C05459=1092.493,135.328,434.820,176.042,18.380,152.701
C05460=1092.487,135.079,434.840,176.041,18.379,152.701
C05461=1092.482,134.830,434.859,176.038,18.378,152.701
C05462=1092.476,134.580,434.880,176.035,18.377,152.702
C05463=1092.470,134.332,434.900,176.032,18.376,152.702
C05464=1092.465,134.082,434.919,176.030,18.376,152.702
C05465=1092.459,133.833,434.940,176.027,18.375,152.703
C05466=1092.454,133.585,434.959,176.025,18.374,152.703
C05467=1092.449,133.335,434.979,176.022,18.372,152.703
C05468=1092.443,133.086,434.999,176.020,18.372,152.703
C05469=1092.437,132.837,435.018,176.017,18.371,152.704
C05470=1092.432,132.588,435.039,176.015,18.370,152.704
C05471=1092.426,132.338,435.058,176.012,18.368,152.704
C05472=1092.420,132.090,435.078,176.010,18.368,152.704
C05473=1092.415,131.841,435.099,176.007,18.367,152.705
C05474=1092.409,131.591,435.118,176.004,18.366,152.705
C05475=1092.403,131.342,435.138,176.001,18.365,152.705
C05476=1092.398,131.093,435.157,175.999,18.364,152.706
C05477=1092.392,130.844,435.177,175.997,18.363,152.706
C05478=1092.386,130.595,435.196,175.994,18.362,152.706
C05479=1092.381,130.345,435.217,175.992,18.361,152.706
C05480=1092.375,130.096,435.236,175.989,18.360,152.707
C05481=1092.369,129.847,435.256,175.987,18.359,152.707
C05482=1092.363,129.598,435.275,175.984,18.358,152.707
C05483=1092.358,129.349,435.295,175.982,18.357,152.707
C05484=1092.352,129.100,435.314,175.979,18.356,152.708
C05485=1092.347,128.850,435.335,175.976,18.355,152.708
C05486=1092.341,128.601,435.354,175.975,18.355,152.708
C05487=1092.335,128.352,435.374,175.972,18.353,152.708
C05488=1092.328,128.076,435.395,175.969,18.352,152.709
C05489=1092.322,127.799,435.418,175.966,18.352,152.709
C05490=1092.316,127.522,435.439,175.963,18.351,152.709
C05491=1092.310,127.246,435.460,175.961,18.349,152.710
C05492=1092.304,126.997,435.480,175.958,18.348,152.710
C05493=1092.298,126.748,435.499,175.955,18.347,152.710
C05494=1092.292,126.499,435.519,175.953,18.347,152.710
C05495=1092.287,126.249,435.539,175.950,18.345,152.711
C05496=1092.282,126.000,435.558,175.948,18.344,152.711
C05497=1092.276,125.751,435.578,175.946,18.344,152.711
C05498=1092.270,125.502,435.597,175.943,18.343,152.711
C05499=1092.265,125.253,435.617,175.940,18.341,152.712
C05500=1092.259,125.003,435.636,175.938,18.340,152.712
C05501=1092.253,124.754,435.656,175.936,18.339,152.712
C05502=1092.247,124.505,435.675,175.933,18.338,152.712
C05503=1092.242,124.255,435.694,175.930,18.337,152.713
C05504=1092.236,124.007,435.714,175.928,18.336,152.713
C05505=1092.231,123.758,435.733,175.926,18.335,152.713
C05506=1092.225,123.508,435.752,175.923,18.334,152.713
C05507=1092.219,123.259,435.772,175.920,18.333,152.714
C05508=1092.214,123.010,435.791,175.918,18.332,152.714
C05509=1092.208,122.760,435.811,175.916,18.331,152.714
C05510=1092.203,122.512,435.830,175.913,18.330,152.714
C05511=1092.198,122.262,435.849,175.911,18.329,152.715
C05512=1092.192,122.013,435.869,175.908,18.328,152.715
C05513=1092.186,121.763,435.888,175.906,18.327,152.715
C05514=1092.180,121.515,435.908,175.904,18.326,152.715
C05515=1092.175,121.266,435.927,175.901,18.324,152.715
C05516=1092.169,121.016,435.946,175.899,18.323,152.716
C05517=1092.164,120.767,435.965,175.897,18.323,152.716
C05518=1092.158,120.518,435.985,175.894,18.322,152.716
C05519=1092.152,120.268,436.004,175.891,18.320,152.716
C05520=1092.147,120.019,436.023,175.890,18.319,152.717
C05521=1092.142,119.770,436.042,175.887,18.318,152.717
C05522=1092.136,119.521,436.062,175.884,18.317,152.717
C05523=1092.130,119.272,436.081,175.881,18.316,152.717
C05524=1092.125,119.023,436.100,175.880,18.315,152.717
C05525=1092.119,118.774,436.119,175.877,18.314,152.718
C05526=1092.113,118.524,436.138,175.874,18.313,152.718
C05527=1092.108,118.275,436.157,175.872,18.312,152.718
C05528=1092.103,118.026,436.177,175.870,18.310,152.718
C05529=1092.097,117.777,436.196,175.867,18.309,152.719
C05530=1092.091,117.527,436.214,175.865,18.309,152.719
C05531=1092.085,117.279,436.233,175.863,18.307,152.719
C05532=1092.080,117.029,436.253,175.860,18.306,152.719
C05533=1092.074,116.780,436.272,175.858,18.305,152.719
C05534=1092.069,116.531,436.291,175.855,18.304,152.720
C05535=1092.063,116.282,436.310,175.853,18.303,152.720
C05536=1092.058,116.032,436.329,175.851,18.302,152.720
C05537=1092.053,115.784,436.348,175.848,18.300,152.720
C05538=1092.047,115.534,436.367,175.846,18.299,152.721
C05539=1092.041,115.284,436.386,175.844,18.299,152.721
C05540=1092.036,115.035,436.405,175.841,18.297,152.721
C05541=1092.031,114.786,436.424,175.838,18.296,152.721
C05542=1092.025,114.536,436.443,175.837,18.295,152.721
C05543=1092.019,114.288,436.461,175.834,18.294,152.722
C05544=1092.013,114.039,436.481,175.831,18.293,152.722
C05545=1092.008,113.789,436.500,175.829,18.292,152.722
C05546=1092.003,113.540,436.519,175.827,18.290,152.722
C05547=1091.997,113.291,436.537,175.824,18.289,152.722
C05548=1091.991,113.041,436.556,175.822,18.289,152.723
C05549=1091.986,112.793,436.575,175.820,18.287,152.723
C05550=1091.980,112.543,436.594,175.817,18.286,152.723
C05551=1091.974,112.294,436.613,175.815,18.285,152.723
C05552=1091.968,112.017,436.634,175.813,18.284,152.723
C05553=1091.962,111.741,436.654,175.810,18.283,152.724
C05554=1091.956,111.465,436.676,175.807,18.281,152.724
C05555=1091.949,111.187,436.696,175.805,18.280,152.724
C05556=1091.943,110.939,436.715,175.802,18.279,152.724
C05557=1091.938,110.690,436.734,175.800,18.278,152.725
C05558=1091.932,110.439,436.752,175.798,18.276,152.725
C05559=1091.926,110.191,436.771,175.795,18.275,152.725
C05560=1091.921,109.942,436.790,175.793,18.274,152.725
C05561=1091.915,109.692,436.809,175.790,18.273,152.725
C05562=1091.910,109.443,436.827,175.788,18.272,152.726
C05563=1091.904,109.194,436.846,175.786,18.271,152.726
C05564=1091.898,108.945,436.864,175.783,18.270,152.726
C05565=1091.893,108.695,436.883,175.781,18.268,152.726
C05566=1091.887,108.446,436.902,175.779,18.268,152.726
C05567=1091.881,108.197,436.920,175.776,18.266,152.727
C05568=1091.876,107.947,436.939,175.774,18.265,152.727
C05569=1091.869,107.698,436.958,175.772,18.264,152.727
C05570=1091.865,107.449,436.976,175.769,18.263,152.727
C05571=1091.858,107.200,436.994,175.767,18.262,152.727
C05572=1091.853,106.951,437.013,175.765,18.260,152.727
C05573=1091.848,106.701,437.032,175.762,18.259,152.728
C05574=1091.842,106.453,437.050,175.760,18.258,152.728
C05575=1091.836,106.203,437.069,175.758,18.257,152.728
C05576=1091.830,105.953,437.087,175.755,18.255,152.728
C05577=1091.825,105.705,437.106,175.753,18.255,152.728
C05578=1091.819,105.455,437.124,175.751,18.253,152.729
C05579=1091.814,105.206,437.143,175.749,18.253,152.729
C05580=1091.808,104.956,437.161,175.746,18.251,152.729
C05581=1091.803,104.708,437.180,175.744,18.250,152.729
C05582=1091.797,104.458,437.198,175.742,18.249,152.729
C05583=1091.791,104.209,437.217,175.739,18.248,152.730
C05584=1091.786,103.959,437.235,175.737,18.246,152.730
C05585=1091.780,103.711,437.253,175.735,18.245,152.730
C05586=1091.775,103.461,437.272,175.732,18.244,152.730
C05587=1091.769,103.212,437.290,175.730,18.243,152.730
C05588=1091.764,102.962,437.309,175.728,18.242,152.730
C05589=1091.758,102.714,437.327,175.726,18.240,152.731
C05590=1091.752,102.464,437.345,175.724,18.239,152.731
C05591=1091.746,102.215,437.364,175.721,18.238,152.731
C05592=1091.741,101.965,437.382,175.718,18.237,152.731
C05593=1091.736,101.716,437.400,175.717,18.236,152.731
C05594=1091.730,101.467,437.419,175.714,18.234,152.731
C05595=1091.724,101.218,437.437,175.712,18.233,152.732
C05596=1091.718,100.969,437.455,175.710,18.232,152.732
C05597=1091.713,100.719,437.473,175.707,18.231,152.732
C05598=1091.707,100.470,437.491,175.705,18.229,152.732
C05599=1091.701,100.221,437.510,175.703,18.228,152.732
C05600=1091.696,99.971,437.528,175.701,18.227,152.733
C05601=1091.690,99.722,437.546,175.699,18.226,152.733
C05602=1091.684,99.473,437.564,175.696,18.225,152.733
C05603=1091.679,99.224,437.583,175.694,18.223,152.733
C05604=1091.673,98.974,437.601,175.691,18.222,152.733
C05605=1091.667,98.725,437.619,175.690,18.221,152.733
C05606=1091.662,98.475,437.637,175.687,18.220,152.733
C05607=1091.656,98.226,437.655,175.685,18.219,152.734
C05608=1091.650,97.977,437.674,175.683,18.217,152.734
C05609=1091.644,97.728,437.691,175.680,18.216,152.734
C05610=1091.639,97.478,437.710,175.678,18.215,152.734
C05611=1091.633,97.230,437.728,175.676,18.214,152.734
C05612=1091.627,96.980,437.746,175.673,18.212,152.735
C05613=1091.622,96.731,437.764,175.672,18.211,152.735
C05614=1091.617,96.482,437.782,175.669,18.210,152.735
C05615=1091.611,96.232,437.800,175.667,18.209,152.735
C05616=1091.604,95.955,437.820,175.665,18.208,152.735
C05617=1091.598,95.679,437.840,175.662,18.206,152.735
C05618=1091.592,95.403,437.860,175.659,18.205,152.736
C05619=1091.586,95.126,437.879,175.657,18.203,152.736
C05620=1091.580,94.876,437.898,175.655,18.202,152.736
C05621=1091.574,94.628,437.916,175.653,18.200,152.736
C05622=1091.568,94.378,437.934,175.650,18.199,152.736
C05623=1091.563,94.129,437.952,175.648,18.198,152.736
C05624=1091.558,93.880,437.970,175.646,18.197,152.736
C05625=1091.552,93.630,437.988,175.644,18.196,152.737
C05626=1091.546,93.381,438.005,175.642,18.194,152.737
C05627=1091.541,93.132,438.023,175.639,18.193,152.737
C05628=1091.535,92.882,438.041,175.637,18.192,152.737
C05629=1091.530,92.633,438.060,175.635,18.190,152.737
C05630=1091.524,92.384,438.077,175.633,18.190,152.737
C05631=1091.518,92.135,438.095,175.631,18.188,152.738
C05632=1091.512,91.886,438.113,175.628,18.186,152.738
C05633=1091.507,91.637,438.130,175.626,18.185,152.738
C05634=1091.502,91.386,438.149,175.624,18.184,152.738
C05635=1091.496,91.137,438.166,175.622,18.183,152.738
C05636=1091.491,90.888,438.184,175.620,18.181,152.738
C05637=1091.484,90.639,438.202,175.618,18.180,152.738
C05638=1091.479,90.390,438.219,175.615,18.179,152.738
C05639=1091.473,90.140,438.237,175.613,18.178,152.739
C05640=1091.467,89.891,438.255,175.611,18.177,152.739
C05641=1091.462,89.642,438.272,175.609,18.175,152.739
C05642=1091.456,89.392,438.290,175.607,18.174,152.739
C05643=1091.450,89.143,438.308,175.604,18.173,152.739
C05644=1091.445,88.894,438.325,175.602,18.172,152.739
C05645=1091.438,88.644,438.343,175.600,18.170,152.740
C05646=1091.433,88.395,438.361,175.598,18.168,152.740
C05647=1091.427,88.146,438.379,175.596,18.167,152.740
C05648=1091.421,87.896,438.396,175.593,18.166,152.740
C05649=1091.416,87.647,438.414,175.591,18.165,152.740
C05650=1091.411,87.398,438.431,175.589,18.163,152.740
C05651=1091.404,87.148,438.449,175.587,18.162,152.740
C05652=1091.399,86.899,438.466,175.585,18.161,152.740
C05653=1091.393,86.650,438.484,175.582,18.159,152.741
C05654=1091.387,86.400,438.502,175.580,18.159,152.741
C05655=1091.382,86.151,438.519,175.578,18.157,152.741
C05656=1091.376,85.902,438.537,175.576,18.156,152.741
C05657=1091.371,85.653,438.555,175.574,18.154,152.741
C05658=1091.365,85.403,438.572,175.572,18.153,152.741
C05659=1091.359,85.154,438.589,175.570,18.152,152.741
C05660=1091.354,84.905,438.607,175.568,18.150,152.742
C05661=1091.348,84.656,438.625,175.566,18.149,152.742
C05662=1091.342,84.406,438.642,175.563,18.148,152.742
C05663=1091.337,84.156,438.659,175.561,18.147,152.742
C05664=1091.332,83.907,438.677,175.559,18.145,152.742
C05665=1091.325,83.658,438.694,175.557,18.144,152.742
C05666=1091.319,83.409,438.712,175.555,18.142,152.742
C05667=1091.314,83.159,438.729,175.553,18.141,152.742
C05668=1091.308,82.910,438.746,175.550,18.140,152.743
C05669=1091.303,82.661,438.764,175.549,18.139,152.743
C05670=1091.297,82.411,438.782,175.546,18.137,152.743
C05671=1091.292,82.161,438.799,175.544,18.135,152.743
C05672=1091.286,81.912,438.816,175.542,18.134,152.743
C05673=1091.281,81.663,438.834,175.540,18.133,152.743
C05674=1091.275,81.414,438.851,175.538,18.132,152.743
C05675=1091.270,81.165,438.868,175.536,18.130,152.743
C05676=1091.263,80.915,438.885,175.534,18.129,152.743
C05677=1091.258,80.666,438.902,175.531,18.127,152.744
C05678=1091.252,80.417,438.920,175.530,18.126,152.744
C05679=1091.247,80.168,438.937,175.527,18.125,152.744
C05680=1091.240,79.891,438.957,175.525,18.123,152.744
C05681=1091.234,79.615,438.975,175.522,18.121,152.744
C05682=1091.228,79.338,438.995,175.521,18.120,152.744
C05683=1091.222,79.062,439.013,175.518,18.119,152.744
C05684=1091.216,78.812,439.031,175.516,18.117,152.744
C05685=1091.210,78.563,439.049,175.514,18.116,152.745
C05686=1091.205,78.313,439.066,175.512,18.114,152.745
C05687=1091.199,78.064,439.083,175.510,18.113,152.745
C05688=1091.193,77.815,439.100,175.507,18.112,152.745
C05689=1091.188,77.566,439.117,175.506,18.110,152.745
C05690=1091.183,77.316,439.134,175.503,18.109,152.745
C05691=1091.176,77.067,439.151,175.502,18.108,152.745
C05692=1091.171,76.817,439.168,175.499,18.106,152.745
C05693=1091.165,76.568,439.186,175.497,18.105,152.745
C05694=1091.159,76.319,439.202,175.495,18.103,152.746
C05695=1091.154,76.069,439.220,175.493,18.102,152.746
C05696=1091.148,75.820,439.236,175.491,18.101,152.746
C05697=1091.142,75.570,439.254,175.488,18.099,152.746
C05698=1091.136,75.321,439.271,175.487,18.098,152.746
C05699=1091.131,75.072,439.288,175.484,18.096,152.746
C05700=1091.125,74.822,439.304,175.483,18.095,152.746
C05701=1091.119,74.573,439.322,175.480,18.094,152.746
C05702=1091.114,74.324,439.339,175.478,18.093,152.746
C05703=1091.108,74.075,439.356,175.476,18.091,152.746
C05704=1091.103,73.825,439.373,175.475,18.089,152.747
C05705=1091.097,73.576,439.390,175.472,18.088,152.747
C05706=1091.091,73.326,439.407,175.470,18.087,152.747
C05707=1091.085,73.076,439.424,175.468,18.085,152.747
C05708=1091.080,72.827,439.441,175.466,18.084,152.747
C05709=1091.074,72.578,439.458,175.464,18.082,152.747
C05710=1091.068,72.329,439.475,175.462,18.081,152.747
C05711=1091.062,72.080,439.491,175.460,18.080,152.747
C05712=1091.057,71.830,439.508,175.458,18.078,152.747
C05713=1091.052,71.581,439.526,175.456,18.077,152.747
C05714=1091.046,71.332,439.542,175.454,18.075,152.748
C05715=1091.041,71.082,439.559,175.452,18.074,152.748
C05716=1091.034,70.833,439.576,175.450,18.073,152.748
C05717=1091.029,70.584,439.593,175.448,18.071,152.748
C05718=1091.024,70.334,439.610,175.446,18.070,152.748
C05719=1091.018,70.085,439.626,175.444,18.068,152.748
C05720=1091.012,69.836,439.643,175.442,18.067,152.748
C05721=1091.006,69.586,439.660,175.440,18.065,152.748
C05722=1091.001,69.336,439.677,175.438,18.064,152.748
C05723=1090.994,69.087,439.694,175.435,18.063,152.748
C05724=1090.989,68.837,439.711,175.434,18.061,152.749
C05725=1090.983,68.588,439.727,175.431,18.060,152.749
C05726=1090.978,68.338,439.744,175.430,18.058,152.749
C05727=1090.972,68.090,439.761,175.427,18.057,152.749
C05728=1090.967,67.840,439.778,175.426,18.056,152.749
C05729=1090.961,67.591,439.794,175.423,18.054,152.749
C05730=1090.955,67.341,439.810,175.422,18.053,152.749
C05731=1090.949,67.092,439.827,175.419,18.051,152.749
C05732=1090.943,66.843,439.844,175.418,18.050,152.749
C05733=1090.938,66.593,439.861,175.415,18.048,152.749
C05734=1090.932,66.344,439.877,175.414,18.047,152.749
C05735=1090.927,66.094,439.894,175.411,18.045,152.749
C05736=1090.921,65.845,439.910,175.410,18.044,152.750
C05737=1090.915,65.596,439.926,175.407,18.042,152.750
C05738=1090.909,65.347,439.944,175.406,18.041,152.750
C05739=1090.903,65.097,439.960,175.403,18.039,152.750
C05740=1090.898,64.848,439.977,175.402,18.038,152.750
C05741=1090.892,64.598,439.993,175.399,18.036,152.750
C05742=1090.886,64.349,440.010,175.398,18.035,152.750
C05743=1090.881,64.099,440.026,175.395,18.034,152.750
C05744=1090.874,63.823,440.045,175.394,18.033,152.750
C05745=1090.867,63.546,440.063,175.391,18.031,152.750
C05746=1090.862,63.270,440.081,175.389,18.029,152.750
C05747=1090.855,62.994,440.099,175.386,18.027,152.750
C05748=1090.850,62.744,440.116,175.385,18.026,152.751
C05749=1090.844,62.495,440.132,175.382,18.024,152.751
C05750=1090.838,62.245,440.148,175.381,18.023,152.751
C05751=1090.832,61.996,440.164,175.378,18.022,152.751
C05752=1090.826,61.747,440.181,175.377,18.020,152.751
C05753=1090.821,61.497,440.198,175.374,18.019,152.751
C05754=1090.815,61.248,440.214,175.373,18.017,152.751
C05755=1090.809,60.998,440.230,175.371,18.016,152.751
C05756=1090.803,60.749,440.246,175.369,18.014,152.751
C05757=1090.797,60.499,440.263,175.367,18.013,152.751
C05758=1090.792,60.250,440.279,175.365,18.012,152.751
C05759=1090.786,60.000,440.296,175.363,18.011,152.751
C05760=1090.780,59.751,440.312,175.360,18.009,152.752
C05761=1090.774,59.502,440.328,175.359,18.007,152.752
C05762=1090.768,59.252,440.344,175.357,18.006,152.752
C05763=1090.762,59.003,440.361,175.355,18.005,152.752
C05764=1090.757,58.753,440.378,175.353,18.003,152.752
C05765=1090.751,58.504,440.394,175.351,18.001,152.752
C05766=1090.745,58.255,440.410,175.349,18.000,152.752
C05767=1090.739,58.005,440.426,175.347,17.999,152.752
C05768=1090.733,57.756,440.443,175.345,17.997,152.752
C05769=1090.728,57.507,440.458,175.343,17.996,152.752
C05770=1090.723,57.257,440.475,175.341,17.994,152.752
C05771=1090.717,57.008,440.491,175.339,17.992,152.752
C05772=1090.711,56.758,440.507,175.338,17.991,152.752
C05773=1090.705,56.509,440.523,175.335,17.990,152.752
C05774=1090.699,56.260,440.540,175.334,17.988,152.752
C05775=1090.693,56.010,440.556,175.331,17.986,152.753
C05776=1090.688,55.760,440.571,175.330,17.985,152.753
C05777=1090.682,55.511,440.588,175.327,17.983,152.753
C05778=1090.677,55.262,440.604,175.326,17.982,152.753
C05779=1090.671,55.013,440.620,175.323,17.981,152.753
C05780=1090.665,54.763,440.637,175.322,17.979,152.753
C05781=1090.659,54.513,440.652,175.320,17.978,152.753
C05782=1090.653,54.264,440.669,175.318,17.976,152.753
C05783=1090.648,54.015,440.685,175.316,17.975,152.753
C05784=1090.642,53.766,440.701,175.314,17.973,152.753
C05785=1090.637,53.516,440.716,175.312,17.971,152.753
C05786=1090.631,53.267,440.732,175.310,17.970,152.753
C05787=1090.625,53.017,440.749,175.308,17.969,152.753
C05788=1090.620,52.767,440.765,175.306,17.967,152.753
C05789=1090.614,52.518,440.781,175.304,17.966,152.753
C05790=1090.608,52.269,440.797,175.303,17.964,152.753
C05791=1090.602,52.020,440.813,175.301,17.962,152.753
C05792=1090.597,51.770,440.829,175.299,17.961,152.754
C05793=1090.591,51.520,440.845,175.297,17.959,152.754
C05794=1090.585,51.271,440.861,175.295,17.958,152.754
C05795=1090.580,51.022,440.876,175.293,17.956,152.754
C05796=1090.574,50.773,440.893,175.291,17.955,152.754
C05797=1090.568,50.523,440.909,175.289,17.953,152.754
C05798=1090.562,50.273,440.925,175.287,17.952,152.754
C05799=1090.557,50.025,440.940,175.286,17.951,152.754
C05800=1090.551,49.775,440.956,175.283,17.949,152.754
C05801=1090.545,49.525,440.972,175.282,17.947,152.754
C05802=1090.539,49.276,440.988,175.280,17.945,152.754
C05803=1090.534,49.027,441.004,175.278,17.944,152.754
C05804=1090.528,48.777,441.020,175.276,17.942,152.754
C05805=1090.523,48.527,441.035,175.274,17.941,152.754
C05806=1090.517,48.278,441.052,175.272,17.939,152.754
C05807=1090.512,48.029,441.067,175.270,17.938,152.754
C05808=1090.506,47.752,441.085,175.268,17.936,152.754
C05809=1090.499,47.475,441.103,175.266,17.935,152.754
C05810=1090.493,47.198,441.120,175.264,17.933,152.754
C05811=1090.487,46.922,441.138,175.262,17.930,152.754
C05812=1090.481,46.672,441.153,175.260,17.929,152.754
C05813=1090.476,46.423,441.169,175.258,17.927,152.754
C05814=1090.470,46.173,441.185,175.256,17.926,152.754
C05815=1090.464,45.924,441.201,175.255,17.925,152.754
C05816=1090.459,45.675,441.216,175.253,17.923,152.755
C05817=1090.453,45.425,441.232,175.251,17.921,152.755
C05818=1090.447,45.175,441.248,175.249,17.920,152.755
C05819=1090.442,44.926,441.263,175.247,17.918,152.755
C05820=1090.436,44.677,441.279,175.245,17.917,152.755
C05821=1090.431,44.427,441.295,175.243,17.915,152.755
C05822=1090.425,44.178,441.311,175.242,17.913,152.755
C05823=1090.420,43.928,441.326,175.240,17.912,152.755
C05824=1090.414,43.679,441.343,175.238,17.910,152.755
C05825=1090.409,43.429,441.358,175.236,17.909,152.755
C05826=1090.402,43.180,441.373,175.234,17.907,152.755
C05827=1090.396,42.930,441.389,175.232,17.905,152.755
C05828=1090.391,42.681,441.404,175.230,17.904,152.755
C05829=1090.385,42.432,441.420,175.229,17.903,152.755
C05830=1090.380,42.182,441.436,175.227,17.901,152.755
C05831=1090.374,41.933,441.451,175.225,17.899,152.755
C05832=1090.368,41.684,441.467,175.223,17.897,152.755
C05833=1090.362,41.434,441.482,175.221,17.896,152.755
C05834=1090.357,41.184,441.498,175.220,17.895,152.755
C05835=1090.351,40.935,441.514,175.217,17.893,152.755
C05836=1090.345,40.685,441.529,175.216,17.892,152.755
C05837=1090.340,40.436,441.544,175.213,17.890,152.755
C05838=1090.334,40.187,441.560,175.212,17.888,152.755
C05839=1090.328,39.937,441.576,175.211,17.887,152.755
C05840=1090.322,39.688,441.590,175.208,17.885,152.755
C05841=1090.317,39.438,441.606,175.207,17.884,152.755
C05842=1090.312,39.189,441.622,175.204,17.882,152.755
C05843=1090.306,38.939,441.637,175.203,17.880,152.755
C05844=1090.299,38.690,441.652,175.201,17.879,152.755
C05845=1090.294,38.440,441.667,175.199,17.877,152.755
C05846=1090.288,38.191,441.684,175.198,17.876,152.755
C05847=1090.283,37.942,441.699,175.195,17.874,152.756
C05848=1090.277,37.692,441.714,175.194,17.872,152.756
C05849=1090.271,37.442,441.729,175.192,17.871,152.756
C05850=1090.266,37.193,441.744,175.190,17.869,152.756
C05851=1090.260,36.944,441.760,175.188,17.868,152.756
C05852=1090.254,36.694,441.776,175.186,17.866,152.756
C05853=1090.248,36.445,441.790,175.184,17.865,152.756
C05854=1090.243,36.195,441.806,175.183,17.863,152.756
C05855=1090.236,35.945,441.821,175.181,17.861,152.756
C05856=1090.231,35.697,441.837,175.179,17.860,152.756
C05857=1090.224,35.447,441.852,175.177,17.858,152.756
C05858=1090.219,35.198,441.867,175.175,17.857,152.756
C05859=1090.214,34.948,441.882,175.174,17.855,152.756
C05860=1090.207,34.698,441.897,175.171,17.854,152.756
C05861=1090.202,34.449,441.912,175.170,17.852,152.756
C05862=1090.196,34.199,441.927,175.169,17.851,152.756
C05863=1090.191,33.950,441.943,175.166,17.849,152.756
C05864=1090.184,33.701,441.958,175.165,17.847,152.756
C05865=1090.179,33.452,441.973,175.162,17.846,152.756
C05866=1090.174,33.202,441.989,175.161,17.844,152.756
C05867=1090.167,32.952,442.004,175.160,17.843,152.756
C05868=1090.162,32.703,442.019,175.157,17.841,152.756
C05869=1090.156,32.453,442.034,175.156,17.839,152.756
C05870=1090.151,32.204,442.049,175.154,17.838,152.756
C05871=1090.144,31.954,442.064,175.152,17.836,152.756
C05872=1090.138,31.677,442.081,175.150,17.834,152.756
C05873=1090.132,31.400,442.098,175.148,17.833,152.756
C05874=1090.126,31.124,442.114,175.146,17.831,152.756
C05875=1090.120,30.847,442.131,175.144,17.829,152.756
C05876=1090.113,30.598,442.146,175.142,17.827,152.756
C05877=1090.108,30.348,442.161,175.141,17.826,152.756
C05878=1090.102,30.099,442.176,175.138,17.824,152.756
C05879=1090.097,29.849,442.191,175.137,17.823,152.756
C05880=1090.090,29.600,442.206,175.135,17.821,152.756
C05881=1090.085,29.351,442.221,175.133,17.819,152.756
C05882=1090.079,29.101,442.236,175.131,17.818,152.756
C05883=1090.074,28.852,442.252,175.130,17.816,152.756
C05884=1090.068,28.602,442.266,175.128,17.814,152.756
C05885=1090.063,28.353,442.282,175.126,17.813,152.756
C05886=1090.056,28.103,442.297,175.125,17.812,152.756
C05887=1090.051,27.853,442.310,175.123,17.810,152.756
C05888=1090.045,27.604,442.326,175.121,17.808,152.757
C05889=1090.039,27.355,442.341,175.119,17.806,152.757
C05890=1090.033,27.105,442.356,175.117,17.805,152.756
C05891=1090.028,26.856,442.371,175.116,17.804,152.757
C05892=1090.021,26.606,442.386,175.114,17.802,152.757
C05893=1090.016,26.357,442.401,175.112,17.800,152.756
C05894=1090.010,26.107,442.416,175.110,17.799,152.757
C05895=1090.005,25.857,442.430,175.108,17.797,152.757
C05896=1089.999,25.607,442.445,175.107,17.796,152.757
C05897=1089.993,25.359,442.460,175.105,17.794,152.757
C05898=1089.987,25.109,442.475,175.103,17.792,152.757
C05899=1089.981,24.860,442.489,175.101,17.791,152.757
C05900=1089.975,24.610,442.505,175.100,17.789,152.757
C05901=1089.970,24.360,442.519,175.098,17.787,152.757
C05902=1089.963,24.111,442.534,175.096,17.786,152.757
C05903=1089.958,23.861,442.549,175.095,17.784,152.757
C05904=1089.953,23.613,442.563,175.093,17.782,152.757
C05905=1089.947,23.362,442.578,175.091,17.781,152.757
C05906=1089.941,23.113,442.593,175.090,17.780,152.757
C05907=1089.935,22.863,442.608,175.087,17.778,152.757
C05908=1089.929,22.614,442.622,175.086,17.776,152.757
C05909=1089.923,22.364,442.637,175.084,17.775,152.757
C05910=1089.918,22.115,442.652,175.082,17.773,152.757
C05911=1089.912,21.866,442.666,175.081,17.771,152.757
C05912=1089.906,21.616,442.681,175.078,17.770,152.757
C05913=1089.901,21.366,442.696,175.077,17.768,152.757
C05914=1089.895,21.117,442.711,175.075,17.766,152.757
C05915=1089.889,20.868,442.725,175.073,17.765,152.757
C05916=1089.884,20.618,442.739,175.072,17.763,152.757
C05917=1089.878,20.368,442.755,175.070,17.762,152.757
C05918=1089.872,20.119,442.769,175.068,17.759,152.757
C05919=1089.866,19.869,442.783,175.066,17.758,152.757
C05920=1089.860,19.620,442.798,175.065,17.757,152.757
C05921=1089.855,19.371,442.813,175.063,17.755,152.757
C05922=1089.849,19.121,442.827,175.061,17.754,152.757
C05923=1089.843,18.871,442.842,175.060,17.752,152.757
C05924=1089.837,18.622,442.857,175.058,17.750,152.757
C05925=1089.832,18.372,442.871,175.056,17.749,152.757
C05926=1089.826,18.123,442.885,175.055,17.747,152.757
C05927=1089.820,17.873,442.900,175.053,17.746,152.757
C05928=1089.814,17.624,442.914,175.051,17.744,152.757
C05929=1089.809,17.374,442.928,175.049,17.742,152.757
C05930=1089.803,17.125,442.944,175.048,17.741,152.757
C05931=1089.797,16.876,442.958,175.046,17.739,152.757
C05932=1089.791,16.625,442.972,175.044,17.738,152.757
C05933=1089.785,16.376,442.987,175.043,17.736,152.757
C05934=1089.780,16.127,443.001,175.040,17.734,152.757
C05935=1089.773,15.877,443.016,175.039,17.732,152.757
C05936=1089.768,15.602,443.031,175.037,17.731,152.757
C05937=1089.761,15.326,443.048,175.035,17.729,152.757
C05938=1089.755,15.051,443.063,175.033,17.727,152.757
C05939=1089.748,14.776,443.079,175.032,17.725,152.757
C05940=1089.743,14.527,443.094,175.029,17.723,152.757
C05941=1089.737,14.277,443.108,175.028,17.722,152.757
C05942=1089.731,14.028,443.123,175.026,17.721,152.757
C05943=1089.725,13.778,443.136,175.024,17.719,152.757
C05944=1089.719,13.528,443.151,175.023,17.717,152.757
C05945=1089.713,13.279,443.165,175.021,17.716,152.757
C05946=1089.708,13.029,443.179,175.020,17.714,152.757
C05947=1089.702,12.780,443.194,175.018,17.712,152.757
C05948=1089.696,12.530,443.208,175.016,17.711,152.757
C05949=1089.690,12.281,443.223,175.015,17.709,152.757
C05950=1089.684,12.031,443.237,175.012,17.707,152.757
C05951=1089.679,11.781,443.251,175.011,17.706,152.757
C05952=1089.672,11.533,443.265,175.009,17.705,152.757
C05953=1089.666,11.282,443.279,175.007,17.703,152.757
C05954=1089.660,11.033,443.293,175.006,17.701,152.757
C05955=1089.655,10.784,443.307,175.004,17.700,152.757
C05956=1089.649,10.533,443.322,175.003,17.698,152.757
C05957=1089.643,10.285,443.336,175.001,17.696,152.757
C05958=1089.638,10.035,443.350,174.999,17.695,152.757
C05959=1089.632,9.785,443.364,174.998,17.694,152.757
C05960=1089.626,9.536,443.379,174.995,17.691,152.757
C05961=1089.620,9.286,443.393,174.994,17.690,152.757
C05962=1089.615,9.037,443.407,174.992,17.689,152.757
C05963=1089.608,8.787,443.421,174.990,17.687,152.757
C05964=1089.602,8.538,443.435,174.989,17.685,152.757
C05965=1089.597,8.288,443.449,174.987,17.684,152.757
C05966=1089.591,8.039,443.463,174.986,17.682,152.757
C05967=1089.585,7.789,443.477,174.983,17.680,152.757
C05968=1089.579,7.539,443.491,174.982,17.679,152.757
C05969=1089.574,7.290,443.506,174.980,17.678,152.757
C05970=1089.567,7.041,443.519,174.978,17.675,152.757
C05971=1089.561,6.791,443.533,174.977,17.674,152.757
C05972=1089.556,6.541,443.547,174.975,17.672,152.757
C05973=1089.550,6.292,443.562,174.974,17.671,152.757
C05974=1089.545,6.043,443.576,174.972,17.669,152.757
C05975=1089.538,5.792,443.590,174.970,17.667,152.757
C05976=1089.533,5.543,443.604,174.969,17.666,152.757
C05977=1089.527,5.294,443.617,174.966,17.664,152.757
C05978=1089.521,5.045,443.632,174.965,17.663,152.757
C05979=1089.516,4.795,443.645,174.964,17.661,152.757
C05980=1089.509,4.545,443.660,174.962,17.659,152.757
C05981=1089.504,4.295,443.674,174.960,17.658,152.757
C05982=1089.499,4.046,443.687,174.958,17.656,152.757
C05983=1089.492,3.796,443.701,174.957,17.655,152.757
C05984=1089.487,3.547,443.715,174.955,17.653,152.757
C05985=1089.480,3.297,443.729,174.953,17.651,152.757
C05986=1089.475,3.048,443.743,174.952,17.650,152.757
C05987=1089.469,2.798,443.757,174.950,17.648,152.757
C05988=1089.463,2.549,443.770,174.948,17.646,152.757
C05989=1089.458,2.299,443.784,174.947,17.645,152.757
C05990=1089.452,2.050,443.798,174.945,17.643,152.757
C05991=1089.446,1.799,443.812,174.944,17.642,152.757
C05992=1089.440,1.550,443.827,174.942,17.640,152.757
C05993=1089.434,1.301,443.840,174.940,17.638,152.757
C05994=1089.429,1.051,443.854,174.939,17.637,152.757
C05995=1089.423,0.802,443.868,174.937,17.634,152.757
C05996=1089.418,0.552,443.882,174.935,17.633,152.757
C05997=1089.412,0.303,443.895,174.934,17.632,152.757
C05998=1089.406,0.053,443.909,174.932,17.630,152.757
C05999=1089.400,-0.197,443.923,174.930,17.628,152.757
C06000=1089.395,-0.470,443.938,174.929,17.626,152.757
C06001=1089.388,-0.743,443.953,174.927,17.624,152.757
C06002=1089.381,-1.016,443.969,174.925,17.623,152.757
C06003=1089.375,-1.290,443.984,174.923,17.621,152.757
C06004=1089.369,-1.539,443.997,174.921,17.620,152.757
C06005=1089.364,-1.789,444.011,174.920,17.618,152.757
C06006=1089.358,-2.038,444.025,174.919,17.616,152.757
C06007=1089.352,-2.288,444.038,174.916,17.614,152.757
C06008=1089.347,-2.537,444.052,174.915,17.613,152.757
C06009=1089.341,-2.787,444.066,174.913,17.612,152.757
C06010=1089.336,-3.036,444.080,174.912,17.610,152.757
C06011=1089.329,-3.286,444.093,174.910,17.608,152.757
C06012=1089.323,-3.536,444.107,174.908,17.606,152.757
C06013=1089.317,-3.786,444.120,174.907,17.605,152.757
C06014=1089.312,-4.035,444.134,174.905,17.604,152.757
C06015=1089.306,-4.285,444.147,174.903,17.601,152.757
C06016=1089.300,-4.534,444.161,174.902,17.600,152.757
C06017=1089.295,-4.784,444.175,174.900,17.598,152.757
C06018=1089.289,-5.033,444.188,174.899,17.597,152.757
C06019=1089.283,-5.283,444.202,174.897,17.595,152.757
C06020=1089.276,-5.533,444.215,174.895,17.593,152.757
C06021=1089.271,-5.782,444.229,174.894,17.592,152.757
C06022=1089.265,-6.031,444.243,174.892,17.591,152.757
C06023=1089.259,-6.282,444.256,174.890,17.589,152.757
C06024=1089.253,-6.531,444.269,174.889,17.587,152.757
C06025=1089.248,-6.780,444.283,174.887,17.585,152.757
C06026=1089.242,-7.030,444.296,174.886,17.584,152.757
C06027=1089.236,-7.279,444.310,174.883,17.582,152.757
C06028=1089.230,-7.529,444.323,174.882,17.581,152.757
C06029=1089.225,-7.779,444.336,174.881,17.579,152.757
C06030=1089.218,-8.028,444.350,174.879,17.578,152.757
C06031=1089.213,-8.278,444.363,174.878,17.576,152.757
C06032=1089.207,-8.527,444.377,174.875,17.574,152.757
C06033=1089.200,-8.777,444.390,174.874,17.573,152.757
C06034=1089.195,-9.027,444.404,174.872,17.572,152.757
C06035=1089.189,-9.276,444.417,174.871,17.570,152.757
C06036=1089.183,-9.526,444.431,174.869,17.568,152.757
C06037=1089.177,-9.775,444.444,174.867,17.566,152.757
C06038=1089.172,-10.025,444.457,174.866,17.565,152.757
C06039=1089.165,-10.275,444.470,174.864,17.564,152.757
C06040=1089.160,-10.524,444.484,174.862,17.561,152.757
C06041=1089.154,-10.773,444.498,174.861,17.560,152.757
C06042=1089.149,-11.024,444.511,174.859,17.558,152.757
C06043=1089.142,-11.273,444.524,174.858,17.557,152.757
C06044=1089.136,-11.522,444.537,174.856,17.556,152.757
C06045=1089.131,-11.772,444.550,174.854,17.553,152.757
C06046=1089.125,-12.022,444.564,174.853,17.552,152.757
C06047=1089.119,-12.271,444.577,174.851,17.550,152.757
C06048=1089.113,-12.520,444.591,174.850,17.549,152.757
C06049=1089.108,-12.771,444.604,174.848,17.547,152.757
C06050=1089.102,-13.020,444.617,174.846,17.546,152.757
C06051=1089.096,-13.269,444.630,174.845,17.544,152.757
C06052=1089.090,-13.519,444.644,174.843,17.543,152.757
C06053=1089.084,-13.769,444.657,174.842,17.541,152.757
C06054=1089.079,-14.019,444.670,174.840,17.539,152.757
C06055=1089.073,-14.267,444.683,174.838,17.538,152.757
C06056=1089.067,-14.517,444.696,174.837,17.536,152.757
C06057=1089.062,-14.767,444.709,174.835,17.535,152.757
C06058=1089.056,-15.016,444.723,174.833,17.533,152.757
C06059=1089.050,-15.266,444.735,174.832,17.531,152.757
C06060=1089.044,-15.516,444.749,174.830,17.530,152.757
C06061=1089.038,-15.765,444.762,174.829,17.528,152.757
C06062=1089.032,-16.015,444.775,174.827,17.527,152.757
C06063=1089.026,-16.264,444.788,174.825,17.525,152.757
C06064=1089.020,-16.537,444.802,174.824,17.523,152.757
C06065=1089.013,-16.808,444.816,174.822,17.522,152.757
C06066=1089.007,-17.080,444.831,174.820,17.520,152.757
C06067=1089.000,-17.351,444.845,174.819,17.518,152.757
C06068=1088.995,-17.601,444.858,174.817,17.517,152.757
C06069=1088.989,-17.850,444.872,174.815,17.515,152.757
C06070=1088.983,-18.100,444.884,174.813,17.514,152.757
C06071=1088.977,-18.349,444.898,174.812,17.512,152.757
C06072=1088.971,-18.599,444.910,174.811,17.510,152.757
C06073=1088.965,-18.849,444.924,174.809,17.509,152.757
C06074=1088.959,-19.099,444.937,174.807,17.507,152.757
C06075=1088.954,-19.347,444.949,174.805,17.506,152.757
C06076=1088.948,-19.597,444.962,174.804,17.504,152.757
C06077=1088.942,-19.846,444.975,174.802,17.503,152.757
C06078=1088.936,-20.097,444.988,174.801,17.501,152.757
C06079=1088.931,-20.346,445.001,174.799,17.499,152.757
C06080=1088.924,-20.596,445.014,174.797,17.498,152.757
C06081=1088.918,-20.846,445.027,174.796,17.496,152.757
C06082=1088.912,-21.095,445.040,174.794,17.495,152.757
C06083=1088.907,-21.345,445.053,174.793,17.493,152.757
C06084=1088.901,-21.594,445.066,174.792,17.492,152.757
C06085=1088.895,-21.844,445.079,174.789,17.490,152.757
C06086=1088.890,-22.093,445.091,174.788,17.488,152.757
C06087=1088.883,-22.343,445.104,174.786,17.487,152.757
C06088=1088.877,-22.592,445.117,174.785,17.485,152.757
C06089=1088.871,-22.842,445.130,174.783,17.484,152.757
C06090=1088.866,-23.092,445.143,174.781,17.482,152.757
C06091=1088.860,-23.342,445.156,174.780,17.480,152.757
C06092=1088.854,-23.591,445.169,174.778,17.479,152.757
C06093=1088.849,-23.840,445.181,174.777,17.478,152.757
C06094=1088.843,-24.090,445.194,174.775,17.476,152.757
C06095=1088.837,-24.339,445.207,174.774,17.475,152.757
C06096=1088.831,-24.589,445.220,174.772,17.472,152.757
C06097=1088.825,-24.839,445.233,174.770,17.471,152.757
C06098=1088.819,-25.089,445.246,174.769,17.470,152.757
C06099=1088.814,-25.338,445.258,174.767,17.468,152.757
C06100=1088.808,-25.588,445.271,174.766,17.467,152.757
C06101=1088.802,-25.838,445.284,174.764,17.465,152.757
C06102=1088.796,-26.087,445.297,174.762,17.463,152.757
C06103=1088.790,-26.337,445.309,174.761,17.462,152.757
C06104=1088.784,-26.587,445.322,174.760,17.460,152.757
C06105=1088.778,-26.835,445.335,174.758,17.459,152.757
C06106=1088.773,-27.085,445.347,174.757,17.457,152.757
C06107=1088.767,-27.335,445.360,174.754,17.455,152.757
C06108=1088.761,-27.585,445.373,174.753,17.454,152.757
C06109=1088.755,-27.834,445.386,174.751,17.453,152.757
C06110=1088.749,-28.084,445.398,174.750,17.451,152.757
C06111=1088.743,-28.333,445.411,174.749,17.449,152.757
C06112=1088.737,-28.583,445.423,174.747,17.448,152.757
C06113=1088.731,-28.833,445.436,174.746,17.447,152.757
C06114=1088.725,-29.082,445.449,174.743,17.445,152.757
C06115=1088.719,-29.332,445.461,174.742,17.444,152.757
C06116=1088.713,-29.582,445.474,174.740,17.442,152.757
C06117=1088.708,-29.831,445.486,174.739,17.440,152.757
C06118=1088.702,-30.081,445.499,174.737,17.439,152.757
C06119=1088.696,-30.330,445.512,174.736,17.438,152.757
C06120=1088.689,-30.580,445.524,174.734,17.436,152.757
C06121=1088.683,-30.830,445.537,174.732,17.434,152.757
C06122=1088.678,-31.079,445.549,174.731,17.433,152.757
C06123=1088.672,-31.329,445.561,174.729,17.431,152.757
C06124=1088.666,-31.579,445.574,174.728,17.430,152.757
C06125=1088.660,-31.829,445.586,174.726,17.429,152.757
C06126=1088.655,-32.077,445.599,174.725,17.427,152.757
C06127=1088.649,-32.327,445.612,174.723,17.425,152.757
C06128=1088.643,-32.599,445.625,174.721,17.424,152.757
C06129=1088.636,-32.869,445.638,174.720,17.422,152.757
C06130=1088.629,-33.140,445.652,174.718,17.420,152.757
C06131=1088.623,-33.411,445.665,174.716,17.418,152.757
C06132=1088.618,-33.661,445.678,174.715,17.417,152.757
C06133=1088.612,-33.910,445.690,174.713,17.416,152.757
C06134=1088.606,-34.160,445.703,174.712,17.414,152.757
C06135=1088.600,-34.409,445.716,174.710,17.413,152.757
C06136=1088.594,-34.659,445.728,174.708,17.411,152.757
C06137=1088.588,-34.908,445.740,174.707,17.409,152.757
C06138=1088.582,-35.158,445.753,174.705,17.408,152.757
C06139=1088.576,-35.407,445.765,174.704,17.407,152.757
C06140=1088.570,-35.657,445.777,174.702,17.405,152.757
C06141=1088.565,-35.907,445.790,174.701,17.404,152.757
C06142=1088.559,-36.157,445.803,174.699,17.402,152.757
C06143=1088.553,-36.406,445.814,174.697,17.400,152.757
C06144=1088.547,-36.656,445.827,174.695,17.399,152.757
C06145=1088.541,-36.906,445.839,174.694,17.398,152.757
C06146=1088.535,-37.155,445.851,174.693,17.396,152.757
C06147=1088.530,-37.405,445.864,174.691,17.395,152.757
C06148=1088.524,-37.655,445.877,174.690,17.393,152.757
C06149=1088.518,-37.904,445.887,174.688,17.392,152.757
C06150=1088.512,-38.154,445.900,174.687,17.391,152.757
C06151=1088.506,-38.404,445.913,174.684,17.389,152.757
C06152=1088.501,-38.653,445.925,174.683,17.387,152.757
C06153=1088.495,-38.903,445.937,174.681,17.386,152.757
C06154=1088.488,-39.153,445.949,174.680,17.384,152.757
C06155=1088.483,-39.402,445.961,174.679,17.383,152.757
C06156=1088.477,-39.652,445.974,174.677,17.382,152.757
C06157=1088.470,-39.901,445.986,174.676,17.380,152.757
C06158=1088.464,-40.151,445.998,174.674,17.379,152.757
C06159=1088.458,-40.400,446.010,174.673,17.377,152.757
C06160=1088.453,-40.650,446.023,174.670,17.375,152.757
C06161=1088.447,-40.900,446.034,174.669,17.374,152.757
C06162=1088.441,-41.149,446.046,174.667,17.372,152.757
C06163=1088.435,-41.399,446.059,174.666,17.371,152.757
C06164=1088.429,-41.649,446.071,174.664,17.370,152.757
C06165=1088.423,-41.898,446.083,174.663,17.368,152.757
C06166=1088.417,-42.148,446.095,174.661,17.367,152.757
C06167=1088.411,-42.398,446.107,174.660,17.365,152.757
C06168=1088.405,-42.647,446.119,174.658,17.364,152.758
C06169=1088.400,-42.897,446.131,174.657,17.363,152.757
C06170=1088.393,-43.147,446.143,174.655,17.361,152.757
C06171=1088.388,-43.396,446.155,174.653,17.360,152.758
C06172=1088.382,-43.646,446.168,174.652,17.358,152.758
C06173=1088.375,-43.896,446.179,174.650,17.357,152.758
C06174=1088.370,-44.145,446.191,174.649,17.355,152.758
C06175=1088.363,-44.395,446.203,174.647,17.354,152.758
C06176=1088.357,-44.644,446.216,174.646,17.353,152.758
C06177=1088.352,-44.894,446.227,174.644,17.351,152.758
C06178=1088.346,-45.144,446.239,174.643,17.350,152.758
C06179=1088.341,-45.393,446.252,174.641,17.348,152.758
C06180=1088.334,-45.643,446.264,174.640,17.347,152.758
C06181=1088.328,-45.893,446.275,174.638,17.345,152.758
C06182=1088.323,-46.142,446.288,174.636,17.344,152.758
C06183=1088.316,-46.392,446.300,174.635,17.342,152.758
C06184=1088.311,-46.641,446.312,174.633,17.341,152.758
C06185=1088.305,-46.891,446.323,174.632,17.339,152.758
C06186=1088.299,-47.141,446.336,174.630,17.338,152.758
C06187=1088.293,-47.390,446.347,174.629,17.337,152.758
C06188=1088.287,-47.640,446.359,174.627,17.335,152.758
C06189=1088.282,-47.890,446.371,174.626,17.334,152.758
C06190=1088.275,-48.139,446.383,174.624,17.333,152.758
C06191=1088.270,-48.389,446.395,174.623,17.331,152.758
C06192=1088.263,-48.660,446.407,174.621,17.329,152.758
C06193=1088.257,-48.932,446.421,174.619,17.328,152.758
C06194=1088.250,-49.203,446.433,174.618,17.326,152.758
C06195=1088.244,-49.474,446.446,174.616,17.325,152.758
C06196=1088.239,-49.723,446.458,174.615,17.324,152.758
C06197=1088.232,-49.974,446.470,174.612,17.322,152.758
C06198=1088.227,-50.223,446.482,174.611,17.320,152.758
C06199=1088.220,-50.472,446.494,174.609,17.319,152.758
C06200=1088.215,-50.723,446.506,174.608,17.318,152.758
C06201=1088.209,-50.972,446.517,174.606,17.316,152.758
C06202=1088.202,-51.221,446.529,174.605,17.315,152.758
C06203=1088.196,-51.471,446.540,174.603,17.313,152.758
C06204=1088.190,-51.721,446.553,174.602,17.312,152.758
C06205=1088.184,-51.971,446.564,174.600,17.311,152.758
C06206=1088.178,-52.220,446.575,174.599,17.310,152.758
C06207=1088.172,-52.470,446.587,174.597,17.308,152.758
C06208=1088.166,-52.719,446.599,174.596,17.307,152.758
C06209=1088.160,-52.969,446.611,174.594,17.306,152.759
C06210=1088.154,-53.219,446.623,174.593,17.304,152.759
C06211=1088.148,-53.468,446.634,174.591,17.303,152.759
C06212=1088.142,-53.718,446.645,174.590,17.302,152.759
C06213=1088.136,-53.967,446.657,174.588,17.301,152.759
C06214=1088.130,-54.218,446.669,174.587,17.299,152.759
C06215=1088.124,-54.466,446.680,174.584,17.297,152.759
C06216=1088.118,-54.717,446.692,174.583,17.296,152.759
C06217=1088.111,-54.966,446.704,174.581,17.295,152.759
C06218=1088.106,-55.216,446.715,174.580,17.294,152.759
C06219=1088.099,-55.466,446.727,174.578,17.292,152.759
C06220=1088.094,-55.715,446.738,174.577,17.291,152.759
C06221=1088.087,-55.965,446.750,174.575,17.289,152.759
C06222=1088.082,-56.215,446.761,174.574,17.288,152.759
C06223=1088.076,-56.465,446.773,174.572,17.287,152.759
C06224=1088.070,-56.714,446.784,174.571,17.286,152.759
C06225=1088.063,-56.964,446.795,174.569,17.284,152.759
C06226=1088.058,-57.213,446.808,174.568,17.283,152.759
C06227=1088.052,-57.463,446.819,174.566,17.282,152.759
C06228=1088.046,-57.712,446.831,174.565,17.280,152.759
C06229=1088.039,-57.962,446.842,174.563,17.279,152.759
C06230=1088.034,-58.212,446.853,174.561,17.277,152.759
C06231=1088.028,-58.462,446.865,174.560,17.276,152.760
C06232=1088.022,-58.711,446.876,174.558,17.275,152.760
C06233=1088.015,-58.961,446.888,174.557,17.274,152.760
C06234=1088.010,-59.210,446.899,174.555,17.273,152.760
C06235=1088.004,-59.461,446.911,174.554,17.271,152.760
C06236=1087.998,-59.709,446.922,174.552,17.270,152.760
C06237=1087.992,-59.960,446.934,174.551,17.268,152.760
C06238=1087.986,-60.209,446.944,174.549,17.267,152.760
C06239=1087.979,-60.459,446.956,174.548,17.266,152.760
C06240=1087.974,-60.709,446.968,174.546,17.265,152.760
C06241=1087.968,-60.959,446.979,174.545,17.263,152.760
C06242=1087.962,-61.208,446.991,174.543,17.262,152.760
C06243=1087.955,-61.458,447.002,174.542,17.261,152.760
C06244=1087.950,-61.707,447.013,174.540,17.260,152.760
C06245=1087.944,-61.956,447.025,174.539,17.258,152.760
C06246=1087.938,-62.207,447.036,174.537,17.257,152.760
C06247=1087.932,-62.456,447.047,174.536,17.255,152.760
C06248=1087.926,-62.706,447.059,174.534,17.254,152.760
C06249=1087.920,-62.955,447.070,174.532,17.253,152.760
C06250=1087.914,-63.205,447.081,174.531,17.252,152.760
C06251=1087.909,-63.455,447.093,174.529,17.251,152.760
C06252=1087.903,-63.704,447.104,174.528,17.249,152.760
C06253=1087.896,-63.954,447.116,174.526,17.248,152.761
C06254=1087.890,-64.204,447.126,174.525,17.247,152.761
C06255=1087.884,-64.454,447.138,174.523,17.245,152.761
C06256=1087.878,-64.726,447.150,174.521,17.244,152.761
C06257=1087.871,-64.998,447.162,174.519,17.242,152.761
C06258=1087.865,-65.271,447.175,174.518,17.241,152.761
C06259=1087.858,-65.544,447.186,174.516,17.240,152.761
C06260=1087.853,-65.793,447.199,174.515,17.238,152.761
C06261=1087.847,-66.043,447.210,174.513,17.237,152.761
C06262=1087.841,-66.293,447.221,174.512,17.235,152.761
C06263=1087.835,-66.543,447.232,174.510,17.234,152.761
C06264=1087.829,-66.792,447.243,174.508,17.233,152.761
C06265=1087.823,-67.042,447.254,174.507,17.232,152.761
C06266=1087.816,-67.291,447.266,174.505,17.231,152.761
C06267=1087.811,-67.541,447.277,174.504,17.230,152.761
C06268=1087.806,-67.791,447.288,174.502,17.228,152.761
C06269=1087.799,-68.041,447.299,174.501,17.227,152.761
C06270=1087.794,-68.290,447.310,174.499,17.225,152.761
C06271=1087.788,-68.540,447.321,174.498,17.224,152.761
C06272=1087.782,-68.790,447.332,174.496,17.223,152.762
C06273=1087.776,-69.039,447.344,174.495,17.221,152.762
C06274=1087.770,-69.288,447.355,174.493,17.220,152.762
C06275=1087.763,-69.539,447.366,174.491,17.219,152.762
C06276=1087.758,-69.788,447.377,174.490,17.218,152.762
C06277=1087.752,-70.038,447.388,174.488,17.217,152.762
C06278=1087.747,-70.287,447.399,174.487,17.216,152.762
C06279=1087.741,-70.538,447.410,174.485,17.214,152.762
C06280=1087.735,-70.787,447.421,174.484,17.213,152.762
C06281=1087.729,-71.036,447.432,174.482,17.212,152.762
C06282=1087.723,-71.287,447.443,174.481,17.210,152.762
C06283=1087.717,-71.536,447.454,174.479,17.209,152.762
C06284=1087.711,-71.786,447.465,174.478,17.208,152.762
C06285=1087.706,-72.035,447.476,174.476,17.206,152.762
C06286=1087.699,-72.285,447.487,174.475,17.205,152.762
C06287=1087.693,-72.535,447.498,174.474,17.205,152.762
C06288=1087.688,-72.784,447.509,174.472,17.203,152.762
C06289=1087.681,-73.035,447.520,174.471,17.202,152.762
C06290=1087.676,-73.284,447.531,174.469,17.201,152.763
C06291=1087.670,-73.534,447.542,174.468,17.199,152.763
C06292=1087.664,-73.783,447.553,174.466,17.198,152.763
C06293=1087.658,-74.033,447.564,174.464,17.197,152.763
C06294=1087.652,-74.283,447.575,174.463,17.196,152.763
C06295=1087.646,-74.532,447.586,174.461,17.194,152.763
C06296=1087.641,-74.782,447.597,174.460,17.193,152.763
C06297=1087.634,-75.032,447.608,174.458,17.192,152.763
C06298=1087.629,-75.281,447.619,174.456,17.191,152.763
C06299=1087.623,-75.531,447.630,174.455,17.190,152.763
C06300=1087.616,-75.781,447.640,174.453,17.189,152.763
C06301=1087.610,-76.030,447.651,174.452,17.187,152.763
C06302=1087.604,-76.280,447.662,174.450,17.186,152.763
C06303=1087.598,-76.530,447.673,174.449,17.185,152.764
C06304=1087.592,-76.779,447.684,174.447,17.184,152.764
C06305=1087.586,-77.029,447.695,174.446,17.183,152.764
C06306=1087.581,-77.279,447.705,174.445,17.182,152.764
C06307=1087.574,-77.529,447.716,174.443,17.181,152.764
C06308=1087.568,-77.778,447.727,174.441,17.180,152.764
C06309=1087.562,-78.028,447.738,174.440,17.178,152.764
C06310=1087.557,-78.277,447.749,174.438,17.177,152.764
C06311=1087.550,-78.528,447.760,174.437,17.176,152.764
C06312=1087.545,-78.777,447.771,174.435,17.175,152.764
C06313=1087.538,-79.026,447.781,174.433,17.174,152.764
C06314=1087.533,-79.276,447.791,174.432,17.172,152.764
C06315=1087.526,-79.526,447.802,174.430,17.171,152.764
C06316=1087.521,-79.776,447.813,174.429,17.170,152.764
C06317=1087.515,-80.025,447.824,174.427,17.169,152.765
C06318=1087.508,-80.275,447.835,174.426,17.168,152.765
C06319=1087.502,-80.525,447.846,174.425,17.167,152.765
C06320=1087.496,-80.799,447.857,174.422,17.166,152.765
C06321=1087.489,-81.074,447.869,174.421,17.164,152.765
C06322=1087.482,-81.349,447.880,174.419,17.163,152.765
C06323=1087.476,-81.624,447.892,174.418,17.162,152.765
C06324=1087.470,-81.873,447.903,174.416,17.161,152.765
C06325=1087.464,-82.123,447.913,174.414,17.160,152.765
C06326=1087.457,-82.373,447.924,174.413,17.159,152.765
C06327=1087.451,-82.622,447.934,174.411,17.158,152.766
C06328=1087.445,-82.872,447.945,174.410,17.157,152.766
C06329=1087.439,-83.122,447.956,174.409,17.156,152.766
C06330=1087.433,-83.372,447.966,174.407,17.155,152.766
C06331=1087.427,-83.621,447.977,174.405,17.154,152.766
C06332=1087.421,-83.871,447.988,174.404,17.153,152.766
C06333=1087.415,-84.121,447.997,174.402,17.152,152.766
C06334=1087.409,-84.371,448.009,174.400,17.151,152.766
C06335=1087.402,-84.620,448.019,174.399,17.149,152.766
C06336=1087.396,-84.869,448.030,174.397,17.148,152.766
C06337=1087.391,-85.119,448.040,174.397,17.147,152.766
C06338=1087.384,-85.369,448.050,174.395,17.146,152.767
C06339=1087.378,-85.619,448.061,174.393,17.145,152.767
C06340=1087.372,-85.869,448.071,174.392,17.144,152.767
C06341=1087.366,-86.118,448.082,174.390,17.143,152.767
C06342=1087.360,-86.368,448.093,174.388,17.142,152.767
C06343=1087.354,-86.618,448.103,174.387,17.141,152.767
C06344=1087.348,-86.868,448.114,174.385,17.140,152.767
C06345=1087.341,-87.117,448.124,174.383,17.139,152.767
C06346=1087.336,-87.367,448.134,174.383,17.138,152.767
C06347=1087.330,-87.616,448.145,174.381,17.137,152.767
C06348=1087.324,-87.866,448.155,174.379,17.136,152.768
C06349=1087.318,-88.116,448.166,174.378,17.135,152.768
C06350=1087.311,-88.366,448.176,174.376,17.134,152.768
C06351=1087.306,-88.615,448.187,174.374,17.133,152.768
C06352=1087.299,-88.865,448.196,174.373,17.132,152.768
C06353=1087.294,-89.114,448.207,174.371,17.131,152.768
C06354=1087.288,-89.364,448.217,174.370,17.130,152.768
C06355=1087.281,-89.614,448.228,174.369,17.129,152.768
C06356=1087.275,-89.864,448.239,174.367,17.128,152.768
C06357=1087.269,-90.114,448.248,174.365,17.127,152.769
C06358=1087.264,-90.363,448.259,174.364,17.126,152.769
C06359=1087.257,-90.613,448.269,174.362,17.125,152.769
C06360=1087.252,-90.862,448.280,174.360,17.123,152.769
C06361=1087.245,-91.112,448.289,174.360,17.123,152.769
C06362=1087.240,-91.362,448.300,174.358,17.122,152.769
C06363=1087.233,-91.612,448.310,174.356,17.121,152.769
C06364=1087.227,-91.862,448.321,174.355,17.120,152.769
C06365=1087.222,-92.112,448.331,174.353,17.119,152.769
C06366=1087.215,-92.361,448.342,174.351,17.117,152.769
C06367=1087.210,-92.610,448.352,174.350,17.116,152.770
C06368=1087.203,-92.860,448.362,174.349,17.116,152.770
C06369=1087.198,-93.110,448.373,174.347,17.115,152.770
C06370=1087.191,-93.360,448.382,174.346,17.114,152.770
C06371=1087.186,-93.610,448.393,174.344,17.113,152.770
C06372=1087.180,-93.859,448.403,174.342,17.111,152.770
C06373=1087.174,-94.109,448.413,174.341,17.110,152.770
C06374=1087.167,-94.359,448.424,174.339,17.109,152.770
C06375=1087.162,-94.609,448.434,174.338,17.109,152.771
C06376=1087.155,-94.858,448.444,174.336,17.108,152.771
C06377=1087.150,-95.108,448.454,174.335,17.107,152.771
C06378=1087.143,-95.357,448.465,174.333,17.106,152.771
C06379=1087.138,-95.607,448.475,174.331,17.105,152.771
C06380=1087.131,-95.857,448.485,174.330,17.104,152.771
C06381=1087.126,-96.107,448.495,174.329,17.103,152.771
C06382=1087.120,-96.357,448.505,174.327,17.102,152.771
C06383=1087.114,-96.606,448.516,174.326,17.101,152.771
C06384=1087.107,-96.883,448.526,174.324,17.100,152.772
C06385=1087.101,-97.160,448.537,174.322,17.099,152.772
C06386=1087.093,-97.437,448.549,174.321,17.098,152.772
C06387=1087.087,-97.714,448.561,174.319,17.097,152.772
C06388=1087.081,-97.964,448.570,174.317,17.096,152.772
C06389=1087.075,-98.213,448.580,174.316,17.095,152.772
C06390=1087.069,-98.463,448.590,174.314,17.094,152.772
C06391=1087.063,-98.713,448.600,174.313,17.093,152.772
C06392=1087.057,-98.962,448.610,174.311,17.092,152.773
C06393=1087.051,-99.212,448.620,174.309,17.092,152.773
C06394=1087.045,-99.461,448.631,174.308,17.091,152.773
C06395=1087.039,-99.711,448.640,174.306,17.090,152.773
C06396=1087.032,-99.962,448.650,174.305,17.089,152.773
C06397=1087.026,-100.211,448.661,174.304,17.088,152.773
C06398=1087.020,-100.461,448.671,174.302,17.087,152.773
C06399=1087.014,-100.711,448.680,174.300,17.086,152.774
C06400=1087.007,-100.960,448.691,174.299,17.085,152.774
C06401=1087.002,-101.210,448.701,174.297,17.084,152.774
C06402=1086.996,-101.460,448.710,174.296,17.084,152.774
C06403=1086.990,-101.710,448.720,174.294,17.083,152.774
C06404=1086.984,-101.959,448.731,174.293,17.082,152.774
C06405=1086.978,-102.209,448.740,174.291,17.081,152.774
C06406=1086.971,-102.459,448.750,174.289,17.080,152.774
C06407=1086.965,-102.708,448.760,174.288,17.080,152.775
C06408=1086.960,-102.958,448.770,174.286,17.079,152.775
C06409=1086.953,-103.208,448.780,174.285,17.078,152.775
C06410=1086.947,-103.458,448.790,174.283,17.077,152.775
C06411=1086.941,-103.707,448.800,174.282,17.077,152.775
C06412=1086.935,-103.957,448.810,174.280,17.075,152.775
C06413=1086.929,-104.207,448.820,174.279,17.074,152.775
C06414=1086.923,-104.457,448.829,174.277,17.073,152.776
C06415=1086.917,-104.706,448.839,174.275,17.073,152.776
C06416=1086.911,-104.956,448.850,174.274,17.072,152.776
C06417=1086.905,-105.206,448.859,174.273,17.071,152.776
C06418=1086.899,-105.455,448.869,174.271,17.070,152.776
C06419=1086.893,-105.705,448.878,174.269,17.069,152.776
C06420=1086.886,-105.955,448.888,174.268,17.068,152.776
C06421=1086.881,-106.205,448.899,174.267,17.068,152.777
C06422=1086.874,-106.454,448.908,174.265,17.067,152.777
C06423=1086.868,-106.704,448.918,174.263,17.066,152.777
C06424=1086.862,-106.954,448.927,174.262,17.065,152.777
C06425=1086.856,-107.204,448.937,174.260,17.065,152.777
C06426=1086.850,-107.454,448.947,174.259,17.064,152.777
C06427=1086.844,-107.703,448.957,174.257,17.063,152.777
C06428=1086.838,-107.953,448.967,174.256,17.062,152.778
C06429=1086.832,-108.203,448.977,174.254,17.062,152.778
C06430=1086.825,-108.452,448.986,174.253,17.061,152.778
C06431=1086.819,-108.702,448.996,174.251,17.060,152.778
C06432=1086.813,-108.952,449.005,174.249,17.059,152.778
C06433=1086.807,-109.202,449.015,174.248,17.058,152.778
C06434=1086.801,-109.452,449.024,174.246,17.058,152.779
C06435=1086.795,-109.700,449.034,174.245,17.057,152.779
C06436=1086.789,-109.950,449.044,174.243,17.056,152.779
C06437=1086.783,-110.200,449.054,174.242,17.056,152.779
C06438=1086.777,-110.450,449.064,174.240,17.055,152.779
C06439=1086.771,-110.700,449.073,174.239,17.054,152.779
C06440=1086.765,-110.949,449.083,174.237,17.053,152.780
C06441=1086.759,-111.199,449.092,174.236,17.052,152.780
C06442=1086.752,-111.449,449.102,174.234,17.052,152.780
C06443=1086.746,-111.699,449.111,174.232,17.051,152.780
C06444=1086.740,-111.949,449.121,174.231,17.050,152.780
C06445=1086.734,-112.198,449.131,174.230,17.050,152.780
C06446=1086.728,-112.448,449.140,174.228,17.049,152.781
C06447=1086.722,-112.698,449.150,174.226,17.048,152.781
C06448=1086.715,-112.970,449.160,174.225,17.047,152.781
C06449=1086.708,-113.241,449.170,174.223,17.046,152.781
C06450=1086.703,-113.513,449.181,174.221,17.045,152.781
C06451=1086.695,-113.785,449.192,174.220,17.045,152.781
C06452=1086.689,-114.035,449.201,174.218,17.044,152.782
C06453=1086.683,-114.285,449.211,174.216,17.044,152.782
C06454=1086.677,-114.534,449.220,174.215,17.042,152.782
C06455=1086.671,-114.784,449.230,174.214,17.042,152.782
C06456=1086.665,-115.034,449.239,174.212,17.041,152.782
C06457=1086.659,-115.283,449.249,174.210,17.041,152.783
C06458=1086.653,-115.533,449.258,174.208,17.040,152.783
C06459=1086.647,-115.783,449.268,174.207,17.040,152.783
C06460=1086.640,-116.032,449.277,174.206,17.039,152.783
C06461=1086.634,-116.282,449.287,174.204,17.038,152.783
C06462=1086.627,-116.532,449.296,174.203,17.037,152.783
C06463=1086.621,-116.782,449.306,174.201,17.037,152.784
C06464=1086.616,-117.031,449.315,174.199,17.036,152.784
C06465=1086.609,-117.281,449.324,174.197,17.035,152.784
C06466=1086.604,-117.531,449.333,174.197,17.035,152.784
C06467=1086.597,-117.781,449.343,174.195,17.034,152.784
C06468=1086.591,-118.031,449.352,174.193,17.033,152.784
C06469=1086.585,-118.280,449.362,174.192,17.033,152.785
C06470=1086.579,-118.530,449.372,174.190,17.032,152.785
C06471=1086.573,-118.780,449.381,174.188,17.031,152.785
C06472=1086.567,-119.029,449.390,174.187,17.030,152.785
C06473=1086.560,-119.279,449.399,174.186,17.030,152.785
C06474=1086.554,-119.528,449.409,174.184,17.030,152.786
C06475=1086.548,-119.779,449.418,174.182,17.029,152.786
C06476=1086.542,-120.029,449.427,174.181,17.029,152.786
C06477=1086.536,-120.278,449.437,174.179,17.027,152.786
C06478=1086.530,-120.528,449.446,174.177,17.027,152.786
C06479=1086.524,-120.777,449.456,174.177,17.026,152.786
C06480=1086.518,-121.027,449.465,174.175,17.026,152.787
C06481=1086.511,-121.277,449.474,174.173,17.025,152.787
C06482=1086.505,-121.527,449.483,174.172,17.025,152.787
C06483=1086.499,-121.777,449.493,174.170,17.024,152.787
C06484=1086.493,-122.027,449.502,174.168,17.023,152.787
C06485=1086.487,-122.276,449.512,174.166,17.022,152.788
C06486=1086.481,-122.526,449.521,174.165,17.022,152.788
C06487=1086.474,-122.776,449.529,174.164,17.021,152.788
C06488=1086.468,-123.025,449.539,174.162,17.021,152.788
C06489=1086.462,-123.275,449.548,174.161,17.021,152.788
C06490=1086.456,-123.525,449.558,174.159,17.020,152.789
C06491=1086.451,-123.775,449.566,174.157,17.019,152.789
C06492=1086.445,-124.025,449.576,174.156,17.019,152.789
C06493=1086.438,-124.274,449.585,174.154,17.018,152.789
C06494=1086.431,-124.524,449.594,174.152,17.017,152.789
C06495=1086.425,-124.774,449.604,174.152,17.017,152.789
C06496=1086.419,-125.024,449.613,174.150,17.016,152.790
C06497=1086.413,-125.273,449.621,174.148,17.016,152.790
C06498=1086.407,-125.523,449.631,174.147,17.016,152.790
C06499=1086.401,-125.773,449.640,174.145,17.015,152.790
C06500=1086.395,-126.023,449.649,174.143,17.014,152.791
C06501=1086.388,-126.272,449.658,174.142,17.014,152.791
C06502=1086.382,-126.521,449.668,174.140,17.013,152.791
C06503=1086.377,-126.772,449.676,174.138,17.012,152.791
C06504=1086.370,-127.022,449.686,174.137,17.012,152.791
C06505=1086.363,-127.271,449.695,174.135,17.012,152.792
C06506=1086.358,-127.522,449.704,174.134,17.011,152.792
C06507=1086.352,-127.771,449.713,174.133,17.011,152.792
C06508=1086.345,-128.029,449.722,174.131,17.010,152.792
C06509=1086.342,-128.286,449.733,174.129,17.009,152.792
C06510=1086.343,-128.542,449.745,174.129,17.006,152.792
C06511=1086.350,-128.795,449.758,174.129,17.002,152.791
C06512=1085.947,-128.817,449.629,174.086,17.114,152.821
C06513=1085.940,-128.563,449.616,174.086,17.118,152.821
C06514=1085.939,-128.308,449.604,174.087,17.121,152.822
C06515=1085.942,-128.050,449.593,174.088,17.122,152.822
C06516=1085.947,-127.793,449.584,174.089,17.122,152.822
C06517=1085.954,-127.544,449.575,174.091,17.123,152.821
C06518=1085.960,-127.293,449.566,174.093,17.124,152.821
C06519=1085.966,-127.043,449.556,174.094,17.124,152.821
C06520=1085.973,-126.794,449.547,174.096,17.125,152.821
C06521=1085.978,-126.544,449.539,174.097,17.126,152.821
C06522=1085.985,-126.294,449.529,174.098,17.126,152.820
C06523=1085.991,-126.045,449.520,174.100,17.126,152.820
C06524=1085.998,-125.795,449.511,174.102,17.127,152.820
C06525=1086.004,-125.545,449.502,174.103,17.127,152.820
C06526=1086.009,-125.296,449.493,174.105,17.128,152.820
C06527=1086.016,-125.046,449.484,174.107,17.128,152.819
C06528=1086.022,-124.796,449.474,174.108,17.129,152.819
C06529=1086.028,-124.546,449.465,174.110,17.130,152.819
C06530=1086.034,-124.296,449.456,174.112,17.130,152.819
C06531=1086.040,-124.046,449.446,174.112,17.131,152.819
C06532=1086.047,-123.797,449.438,174.114,17.131,152.818
C06533=1086.053,-123.547,449.429,174.116,17.132,152.818
C06534=1086.059,-123.297,449.419,174.118,17.133,152.818
C06535=1086.065,-123.047,449.410,174.119,17.133,152.818
C06536=1086.071,-122.798,449.400,174.121,17.134,152.818
C06537=1086.076,-122.548,449.392,174.123,17.134,152.817
C06538=1086.083,-122.298,449.383,174.123,17.135,152.817
C06539=1086.089,-122.049,449.373,174.125,17.136,152.817
C06540=1086.096,-121.799,449.364,174.127,17.136,152.817
C06541=1086.102,-121.549,449.354,174.128,17.137,152.817
C06542=1086.108,-121.299,449.345,174.130,17.137,152.816
C06543=1086.113,-121.050,449.336,174.132,17.138,152.816
C06544=1086.120,-120.800,449.327,174.133,17.138,152.816
C06545=1086.126,-120.550,449.317,174.134,17.139,152.816
C06546=1086.133,-120.300,449.308,174.136,17.140,152.816
C06547=1086.139,-120.051,449.298,174.138,17.141,152.815
C06548=1086.145,-119.801,449.289,174.139,17.141,152.815
C06549=1086.151,-119.550,449.280,174.141,17.142,152.815
C06550=1086.156,-119.301,449.271,174.143,17.143,152.815
C06551=1086.162,-119.052,449.261,174.144,17.143,152.815
C06552=1086.169,-118.802,449.251,174.145,17.144,152.815
C06553=1086.176,-118.552,449.243,174.147,17.144,152.814
C06554=1086.182,-118.302,449.233,174.148,17.145,152.814
C06555=1086.188,-118.053,449.223,174.150,17.145,152.814
C06556=1086.194,-117.803,449.214,174.152,17.147,152.814
C06557=1086.200,-117.553,449.204,174.154,17.147,152.814
C06558=1086.205,-117.303,449.196,174.154,17.148,152.814
C06559=1086.212,-117.054,449.186,174.156,17.148,152.813
C06560=1086.218,-116.804,449.177,174.158,17.149,152.813
C06561=1086.224,-116.554,449.167,174.160,17.150,152.813
C06562=1086.230,-116.304,449.157,174.161,17.150,152.813
C06563=1086.236,-116.054,449.148,174.163,17.151,152.813
C06564=1086.243,-115.805,449.138,174.164,17.152,152.813
C06565=1086.249,-115.555,449.129,174.165,17.152,152.812
C06566=1086.255,-115.305,449.119,174.167,17.153,152.812
C06567=1086.261,-115.055,449.110,174.169,17.154,152.812
C06568=1086.267,-114.806,449.100,174.171,17.155,152.812
C06569=1086.274,-114.557,449.091,174.171,17.155,152.812
C06570=1086.280,-114.307,449.082,174.173,17.156,152.812
C06571=1086.285,-114.057,449.072,174.175,17.157,152.811
C06572=1086.291,-113.807,449.062,174.177,17.158,152.811
C06573=1086.298,-113.535,449.052,174.178,17.158,152.811
C06574=1086.305,-113.262,449.042,174.180,17.159,152.811
C06575=1086.311,-112.991,449.032,174.181,17.160,152.811
C06576=1086.319,-112.719,449.021,174.183,17.160,152.810
C06577=1086.325,-112.469,449.011,174.185,17.161,152.810
C06578=1086.331,-112.219,449.002,174.187,17.162,152.810
C06579=1086.336,-111.969,448.992,174.188,17.162,152.810
C06580=1086.342,-111.719,448.982,174.189,17.164,152.810
C06581=1086.349,-111.469,448.973,174.191,17.165,152.810
C06582=1086.355,-111.220,448.963,174.193,17.165,152.809
C06583=1086.360,-110.970,448.954,174.194,17.166,152.809
C06584=1086.367,-110.721,448.944,174.196,17.166,152.809
C06585=1086.373,-110.471,448.935,174.197,17.167,152.809
C06586=1086.379,-110.221,448.925,174.199,17.168,152.809
C06587=1086.385,-109.972,448.915,174.200,17.168,152.809
C06588=1086.392,-109.722,448.905,174.202,17.170,152.809
C06589=1086.398,-109.472,448.896,174.203,17.171,152.808
C06590=1086.404,-109.222,448.886,174.205,17.171,152.808
C06591=1086.410,-108.973,448.877,174.206,17.172,152.808
C06592=1086.415,-108.723,448.866,174.208,17.173,152.808
C06593=1086.422,-108.473,448.857,174.210,17.173,152.808
C06594=1086.428,-108.223,448.847,174.211,17.174,152.808
C06595=1086.434,-107.973,448.838,174.212,17.175,152.808
C06596=1086.440,-107.724,448.827,174.214,17.176,152.807
C06597=1086.447,-107.474,448.818,174.216,17.177,152.807
C06598=1086.453,-107.224,448.808,174.217,17.178,152.807
C06599=1086.459,-106.975,448.799,174.219,17.178,152.807
C06600=1086.464,-106.724,448.789,174.220,17.179,152.807
C06601=1086.471,-106.475,448.779,174.222,17.180,152.807
C06602=1086.477,-106.226,448.769,174.223,17.181,152.807
C06603=1086.483,-105.976,448.759,174.225,17.182,152.806
C06604=1086.489,-105.726,448.750,174.226,17.182,152.806
C06605=1086.495,-105.476,448.739,174.228,17.183,152.806
C06606=1086.501,-105.226,448.730,174.229,17.184,152.806
C06607=1086.508,-104.977,448.720,174.231,17.185,152.806
C06608=1086.514,-104.727,448.710,174.233,17.186,152.806
C06609=1086.520,-104.477,448.700,174.234,17.186,152.806
C06610=1086.525,-104.227,448.690,174.235,17.188,152.805
C06611=1086.531,-103.977,448.681,174.237,17.188,152.805
C06612=1086.538,-103.728,448.670,174.239,17.189,152.805
C06613=1086.544,-103.478,448.661,174.241,17.190,152.805
C06614=1086.550,-103.228,448.651,174.241,17.191,152.805
C06615=1086.556,-102.978,448.641,174.243,17.192,152.805
C06616=1086.562,-102.729,448.631,174.245,17.192,152.805
C06617=1086.568,-102.479,448.621,174.247,17.194,152.804
C06618=1086.574,-102.229,448.611,174.248,17.195,152.804
C06619=1086.580,-101.980,448.601,174.249,17.195,152.804
C06620=1086.586,-101.730,448.591,174.251,17.196,152.804
C06621=1086.592,-101.480,448.581,174.253,17.197,152.804
C06622=1086.598,-101.230,448.571,174.254,17.198,152.804
C06623=1086.605,-100.981,448.561,174.256,17.199,152.804
C06624=1086.611,-100.731,448.552,174.257,17.199,152.804
C06625=1086.616,-100.481,448.541,174.258,17.201,152.803
C06626=1086.623,-100.232,448.531,174.260,17.202,152.803
C06627=1086.629,-99.982,448.522,174.262,17.202,152.803
C06628=1086.634,-99.732,448.511,174.264,17.203,152.803
C06629=1086.641,-99.483,448.501,174.265,17.204,152.803
C06630=1086.647,-99.233,448.492,174.266,17.205,152.803
C06631=1086.653,-98.984,448.482,174.268,17.206,152.803
C06632=1086.659,-98.734,448.471,174.269,17.207,152.803
C06633=1086.666,-98.484,448.461,174.271,17.208,152.802
C06634=1086.672,-98.234,448.451,174.273,17.209,152.802
C06635=1086.677,-97.984,448.441,174.274,17.209,152.802
C06636=1086.684,-97.734,448.431,174.275,17.210,152.802
C06637=1086.690,-97.458,448.420,174.277,17.211,152.802
C06638=1086.696,-97.181,448.408,174.279,17.213,152.802
C06639=1086.704,-96.903,448.397,174.280,17.214,152.802
C06640=1086.710,-96.626,448.386,174.282,17.215,152.802
C06641=1086.716,-96.376,448.376,174.284,17.216,152.801
C06642=1086.722,-96.127,448.366,174.285,17.217,152.801
C06643=1086.727,-95.877,448.356,174.287,17.218,152.801
C06644=1086.734,-95.628,448.345,174.289,17.219,152.801
C06645=1086.739,-95.378,448.335,174.290,17.220,152.801
C06646=1086.746,-95.129,448.325,174.291,17.221,152.801
C06647=1086.751,-94.878,448.315,174.293,17.221,152.801
C06648=1086.758,-94.629,448.304,174.295,17.222,152.801
C06649=1086.764,-94.378,448.294,174.296,17.223,152.800
C06650=1086.770,-94.129,448.284,174.298,17.224,152.800
C06651=1086.776,-93.879,448.274,174.300,17.226,152.800
C06652=1086.782,-93.629,448.264,174.300,17.226,152.800
C06653=1086.788,-93.380,448.253,174.302,17.227,152.800
C06654=1086.794,-93.130,448.244,174.304,17.228,152.800
C06655=1086.800,-92.881,448.233,174.305,17.229,152.800
C06656=1086.806,-92.631,448.223,174.307,17.230,152.800
C06657=1086.811,-92.381,448.212,174.309,17.231,152.800
C06658=1086.818,-92.131,448.203,174.310,17.233,152.799
C06659=1086.823,-91.882,448.192,174.311,17.233,152.799
C06660=1086.830,-91.631,448.182,174.313,17.234,152.799
C06661=1086.836,-91.382,448.171,174.314,17.235,152.799
C06662=1086.842,-91.133,448.161,174.316,17.236,152.799
C06663=1086.848,-90.883,448.151,174.318,17.237,152.799
C06664=1086.854,-90.634,448.140,174.319,17.238,152.799
C06665=1086.860,-90.383,448.130,174.321,17.240,152.799
C06666=1086.865,-90.134,448.119,174.322,17.241,152.799
C06667=1086.872,-89.884,448.110,174.323,17.242,152.799
C06668=1086.878,-89.634,448.098,174.325,17.243,152.799
C06669=1086.884,-89.385,448.088,174.327,17.244,152.799
C06670=1086.890,-89.135,448.078,174.328,17.245,152.798
C06671=1086.896,-88.885,448.068,174.330,17.246,152.798
C06672=1086.902,-88.635,448.058,174.331,17.247,152.798
C06673=1086.908,-88.386,448.047,174.333,17.248,152.798
C06674=1086.915,-88.136,448.036,174.335,17.249,152.798
C06675=1086.920,-87.886,448.026,174.336,17.250,152.798
C06676=1086.926,-87.637,448.016,174.337,17.251,152.798
C06677=1086.932,-87.387,448.005,174.339,17.252,152.798
C06678=1086.938,-87.137,447.995,174.340,17.253,152.798
C06679=1086.944,-86.888,447.984,174.342,17.254,152.797
C06680=1086.950,-86.637,447.974,174.344,17.255,152.797
C06681=1086.957,-86.388,447.963,174.345,17.256,152.797
C06682=1086.962,-86.138,447.953,174.347,17.257,152.797
C06683=1086.969,-85.889,447.942,174.349,17.258,152.797
C06684=1086.974,-85.639,447.932,174.349,17.260,152.797
C06685=1086.981,-85.389,447.921,174.351,17.261,152.797
C06686=1086.987,-85.140,447.911,174.353,17.262,152.797
C06687=1086.993,-84.890,447.900,174.354,17.263,152.797
C06688=1086.999,-84.641,447.890,174.356,17.264,152.797
C06689=1087.005,-84.391,447.879,174.357,17.265,152.797
C06690=1087.011,-84.140,447.869,174.359,17.266,152.796
C06691=1087.017,-83.891,447.858,174.361,17.267,152.796
C06692=1087.023,-83.642,447.848,174.362,17.268,152.796
C06693=1087.029,-83.392,447.837,174.363,17.269,152.796
C06694=1087.036,-83.142,447.827,174.365,17.270,152.796
C06695=1087.041,-82.892,447.816,174.366,17.271,152.796
C06696=1087.048,-82.643,447.806,174.368,17.272,152.796
C06697=1087.053,-82.393,447.795,174.370,17.274,152.796
C06698=1087.060,-82.143,447.783,174.371,17.275,152.796
C06699=1087.066,-81.893,447.774,174.373,17.276,152.796
C06700=1087.072,-81.644,447.763,174.374,17.277,152.796
C06701=1087.078,-81.369,447.751,174.376,17.278,152.795
C06702=1087.086,-81.094,447.740,174.378,17.279,152.795
C06703=1087.092,-80.819,447.728,174.379,17.281,152.795
C06704=1087.099,-80.544,447.716,174.381,17.282,152.795
C06705=1087.105,-80.295,447.705,174.382,17.283,152.795
C06706=1087.112,-80.045,447.695,174.384,17.284,152.795
C06707=1087.117,-79.796,447.684,174.386,17.285,152.795
C06708=1087.123,-79.545,447.674,174.387,17.286,152.795
C06709=1087.129,-79.296,447.663,174.389,17.288,152.795
C06710=1087.134,-79.046,447.652,174.390,17.289,152.795
C06711=1087.141,-78.797,447.641,174.392,17.290,152.795
C06712=1087.147,-78.547,447.630,174.394,17.291,152.794
C06713=1087.153,-78.298,447.619,174.395,17.292,152.795
C06714=1087.158,-78.048,447.609,174.397,17.293,152.794
C06715=1087.165,-77.797,447.598,174.398,17.294,152.794
C06716=1087.170,-77.548,447.587,174.399,17.295,152.794
C06717=1087.177,-77.299,447.577,174.401,17.297,152.794
C06718=1087.183,-77.048,447.566,174.402,17.298,152.794
C06719=1087.189,-76.799,447.555,174.404,17.299,152.794
C06720=1087.195,-76.549,447.544,174.405,17.300,152.794
C06721=1087.200,-76.300,447.533,174.407,17.302,152.794
C06722=1087.207,-76.050,447.522,174.409,17.303,152.794
C06723=1087.213,-75.801,447.511,174.410,17.304,152.794
C06724=1087.219,-75.551,447.501,174.412,17.305,152.794
C06725=1087.225,-75.301,447.489,174.413,17.306,152.794
C06726=1087.231,-75.051,447.478,174.415,17.307,152.794
C06727=1087.237,-74.801,447.468,174.416,17.309,152.793
C06728=1087.242,-74.552,447.457,174.418,17.310,152.793
C06729=1087.249,-74.302,447.446,174.419,17.311,152.793
C06730=1087.254,-74.052,447.435,174.421,17.312,152.793
C06731=1087.260,-73.803,447.424,174.423,17.313,152.793
C06732=1087.266,-73.552,447.413,174.424,17.315,152.793
C06733=1087.272,-73.303,447.402,174.426,17.316,152.793
C06734=1087.278,-73.054,447.391,174.427,17.317,152.793
C06735=1087.284,-72.804,447.381,174.428,17.318,152.793
C06736=1087.290,-72.554,447.369,174.430,17.319,152.793
C06737=1087.296,-72.304,447.358,174.431,17.320,152.793
C06738=1087.301,-72.055,447.348,174.433,17.322,152.793
C06739=1087.307,-71.805,447.337,174.434,17.323,152.793
C06740=1087.314,-71.555,447.325,174.436,17.325,152.793
C06741=1087.319,-71.306,447.315,174.437,17.326,152.793
C06742=1087.325,-71.057,447.303,174.439,17.327,152.793
C06743=1087.332,-70.807,447.292,174.440,17.328,152.793
C06744=1087.337,-70.557,447.281,174.442,17.329,152.793
C06745=1087.343,-70.308,447.270,174.443,17.331,152.793
C06746=1087.349,-70.058,447.259,174.445,17.332,152.793
C06747=1087.354,-69.808,447.247,174.447,17.333,152.792
C06748=1087.360,-69.558,447.236,174.448,17.335,152.792
C06749=1087.366,-69.309,447.225,174.450,17.336,152.792
C06750=1087.372,-69.058,447.214,174.451,17.337,152.792
C06751=1087.378,-68.809,447.203,174.453,17.339,152.792
C06752=1087.384,-68.560,447.192,174.454,17.340,152.792
C06753=1087.390,-68.310,447.180,174.456,17.341,152.792
C06754=1087.396,-68.060,447.170,174.457,17.342,152.792
C06755=1087.402,-67.811,447.159,174.459,17.344,152.792
C06756=1087.408,-67.561,447.147,174.460,17.345,152.792
C06757=1087.413,-67.311,447.136,174.462,17.346,152.792
C06758=1087.419,-67.061,447.125,174.463,17.348,152.792
C06759=1087.425,-66.811,447.114,174.465,17.349,152.792
C06760=1087.431,-66.562,447.102,174.466,17.350,152.792
C06761=1087.437,-66.313,447.091,174.468,17.351,152.792
C06762=1087.443,-66.063,447.080,174.470,17.353,152.792
C06763=1087.449,-65.813,447.069,174.471,17.354,152.792
C06764=1087.456,-65.563,447.058,174.473,17.355,152.792
C06765=1087.462,-65.291,447.046,174.474,17.357,152.792
C06766=1087.468,-65.018,447.033,174.476,17.358,152.792
C06767=1087.475,-64.745,447.021,174.477,17.359,152.792
C06768=1087.481,-64.473,447.009,174.480,17.361,152.791
C06769=1087.487,-64.223,446.997,174.481,17.363,152.791
C06770=1087.493,-63.974,446.986,174.483,17.364,152.791
C06771=1087.499,-63.724,446.975,174.484,17.365,152.791
C06772=1087.504,-63.474,446.963,174.486,17.366,152.791
C06773=1087.510,-63.224,446.952,174.487,17.368,152.791
C06774=1087.517,-62.975,446.940,174.489,17.369,152.791
C06775=1087.522,-62.725,446.929,174.490,17.370,152.791
C06776=1087.529,-62.475,446.918,174.492,17.372,152.791
C06777=1087.535,-62.226,446.907,174.493,17.373,152.791
C06778=1087.540,-61.976,446.895,174.495,17.374,152.791
C06779=1087.546,-61.726,446.884,174.496,17.376,152.791
C06780=1087.553,-61.476,446.873,174.498,17.377,152.791
C06781=1087.559,-61.227,446.861,174.499,17.378,152.791
C06782=1087.564,-60.978,446.850,174.501,17.379,152.791
C06783=1087.571,-60.728,446.839,174.502,17.381,152.791
C06784=1087.576,-60.478,446.827,174.504,17.382,152.791
C06785=1087.582,-60.228,446.816,174.505,17.384,152.791
C06786=1087.588,-59.979,446.805,174.507,17.385,152.791
C06787=1087.595,-59.729,446.793,174.508,17.386,152.791
C06788=1087.600,-59.479,446.781,174.510,17.387,152.791
C06789=1087.606,-59.229,446.770,174.511,17.389,152.791
C06790=1087.612,-58.980,446.758,174.513,17.390,152.791
C06791=1087.618,-58.730,446.747,174.514,17.392,152.791
C06792=1087.624,-58.481,446.736,174.516,17.393,152.790
C06793=1087.630,-58.231,446.724,174.517,17.394,152.791
C06794=1087.636,-57.981,446.713,174.519,17.395,152.790
C06795=1087.642,-57.732,446.701,174.521,17.396,152.790
C06796=1087.648,-57.482,446.690,174.522,17.398,152.790
C06797=1087.654,-57.232,446.677,174.524,17.399,152.790
C06798=1087.660,-56.983,446.667,174.525,17.401,152.790
C06799=1087.666,-56.733,446.655,174.527,17.402,152.790
C06800=1087.672,-56.484,446.644,174.528,17.403,152.790
C06801=1087.679,-56.233,446.632,174.530,17.404,152.790
C06802=1087.684,-55.984,446.620,174.531,17.406,152.790
C06803=1087.690,-55.734,446.609,174.533,17.407,152.790
C06804=1087.696,-55.485,446.597,174.534,17.409,152.790
C06805=1087.702,-55.235,446.586,174.537,17.410,152.790
C06806=1087.708,-54.985,446.574,174.538,17.412,152.790
C06807=1087.714,-54.736,446.563,174.540,17.413,152.790
C06808=1087.721,-54.486,446.551,174.541,17.415,152.790
C06809=1087.726,-54.236,446.539,174.543,17.416,152.790
C06810=1087.733,-53.987,446.527,174.544,17.417,152.790
C06811=1087.738,-53.737,446.517,174.546,17.418,152.790
C06812=1087.745,-53.488,446.505,174.547,17.420,152.790
C06813=1087.751,-53.237,446.493,174.549,17.421,152.790
C06814=1087.757,-52.988,446.481,174.550,17.423,152.790
C06815=1087.763,-52.739,446.469,174.552,17.424,152.790
C06816=1087.768,-52.489,446.458,174.553,17.425,152.790
C06817=1087.775,-52.239,446.446,174.555,17.426,152.790
C06818=1087.781,-51.989,446.434,174.556,17.428,152.790
C06819=1087.787,-51.740,446.423,174.558,17.429,152.789
C06820=1087.793,-51.490,446.411,174.559,17.431,152.790
C06821=1087.799,-51.241,446.399,174.561,17.432,152.789
C06822=1087.806,-50.991,446.388,174.562,17.433,152.789
C06823=1087.811,-50.741,446.376,174.564,17.434,152.789
C06824=1087.817,-50.492,446.364,174.566,17.437,152.789
C06825=1087.823,-50.241,446.352,174.568,17.438,152.789
C06826=1087.829,-49.993,446.341,174.569,17.439,152.789
C06827=1087.835,-49.743,446.328,174.570,17.441,152.789
C06828=1087.840,-49.493,446.317,174.572,17.442,152.789
C06829=1087.847,-49.222,446.304,174.573,17.443,152.789
C06830=1087.854,-48.950,446.291,174.575,17.445,152.789
C06831=1087.860,-48.679,446.278,174.577,17.447,152.789
C06832=1087.866,-48.408,446.265,174.579,17.448,152.789
C06833=1087.873,-48.158,446.253,174.580,17.450,152.789
C06834=1087.878,-47.908,446.242,174.582,17.451,152.789
C06835=1087.884,-47.659,446.230,174.583,17.453,152.789
C06836=1087.889,-47.410,446.217,174.584,17.454,152.789
C06837=1087.896,-47.159,446.206,174.586,17.455,152.789
C06838=1087.902,-46.909,446.194,174.587,17.457,152.789
C06839=1087.907,-46.660,446.181,174.589,17.458,152.789
C06840=1087.914,-46.411,446.170,174.591,17.460,152.789
C06841=1087.919,-46.161,446.158,174.593,17.462,152.789
C06842=1087.925,-45.911,446.146,174.594,17.463,152.789
C06843=1087.931,-45.661,446.134,174.596,17.464,152.789
C06844=1087.936,-45.412,446.122,174.597,17.466,152.789
C06845=1087.943,-45.162,446.110,174.599,17.467,152.789
C06846=1087.948,-44.913,446.098,174.600,17.469,152.789
C06847=1087.955,-44.663,446.086,174.601,17.470,152.789
C06848=1087.960,-44.413,446.074,174.603,17.471,152.789
C06849=1087.966,-44.164,446.062,174.604,17.473,152.789
C06850=1087.972,-43.914,446.050,174.606,17.474,152.789
C06851=1087.978,-43.664,446.037,174.608,17.476,152.789
C06852=1087.984,-43.415,446.026,174.610,17.478,152.789
C06853=1087.990,-43.165,446.014,174.611,17.479,152.789
C06854=1087.996,-42.915,446.001,174.613,17.480,152.789
C06855=1088.002,-42.666,445.990,174.614,17.482,152.789
C06856=1088.008,-42.416,445.977,174.615,17.483,152.789
C06857=1088.014,-42.167,445.965,174.617,17.485,152.789
C06858=1088.020,-41.917,445.953,174.618,17.486,152.789
C06859=1088.025,-41.667,445.941,174.620,17.488,152.789
C06860=1088.032,-41.417,445.929,174.622,17.489,152.789
C06861=1088.037,-41.168,445.917,174.624,17.491,152.789
C06862=1088.043,-40.918,445.905,174.625,17.493,152.789
C06863=1088.050,-40.669,445.893,174.627,17.494,152.789
C06864=1088.055,-40.420,445.880,174.628,17.495,152.789
C06865=1088.061,-40.170,445.868,174.629,17.497,152.789
C06866=1088.068,-39.920,445.856,174.631,17.498,152.789
C06867=1088.073,-39.670,445.844,174.632,17.499,152.789
C06868=1088.079,-39.420,445.832,174.634,17.501,152.789
C06869=1088.085,-39.171,445.820,174.636,17.503,152.789
C06870=1088.091,-38.921,445.807,174.638,17.504,152.789
C06871=1088.097,-38.672,445.795,174.639,17.506,152.789
C06872=1088.103,-38.422,445.783,174.641,17.507,152.789
C06873=1088.109,-38.172,445.771,174.642,17.509,152.789
C06874=1088.114,-37.923,445.758,174.643,17.510,152.789
C06875=1088.120,-37.673,445.746,174.645,17.511,152.789
C06876=1088.126,-37.423,445.733,174.646,17.513,152.789
C06877=1088.132,-37.175,445.722,174.648,17.514,152.789
C06878=1088.138,-36.925,445.709,174.650,17.517,152.789
C06879=1088.144,-36.675,445.697,174.652,17.518,152.789
C06880=1088.150,-36.425,445.684,174.653,17.519,152.789
C06881=1088.155,-36.176,445.672,174.654,17.521,152.789
C06882=1088.161,-35.926,445.659,174.656,17.522,152.789
C06883=1088.167,-35.676,445.647,174.657,17.523,152.789
C06884=1088.173,-35.427,445.635,174.659,17.525,152.789
C06885=1088.179,-35.177,445.623,174.661,17.527,152.789
C06886=1088.185,-34.927,445.610,174.662,17.529,152.789
C06887=1088.191,-34.677,445.598,174.664,17.530,152.789
C06888=1088.196,-34.428,445.585,174.665,17.531,152.789
C06889=1088.202,-34.178,445.573,174.667,17.533,152.789
C06890=1088.208,-33.928,445.560,174.668,17.535,152.789
C06891=1088.214,-33.680,445.549,174.670,17.536,152.789
C06892=1088.220,-33.430,445.536,174.672,17.538,152.789
C06893=1088.227,-33.159,445.522,174.673,17.539,152.789
C06894=1088.233,-32.887,445.509,174.675,17.541,152.789
C06895=1088.239,-32.617,445.495,174.677,17.543,152.789
C06896=1088.246,-32.346,445.481,174.679,17.544,152.789
C06897=1088.251,-32.096,445.469,174.680,17.546,152.789
C06898=1088.257,-31.847,445.456,174.681,17.547,152.789
C06899=1088.263,-31.597,445.444,174.683,17.549,152.789
C06900=1088.269,-31.347,445.432,174.684,17.550,152.789
C06901=1088.275,-31.097,445.419,174.687,17.552,152.789
C06902=1088.281,-30.847,445.407,174.688,17.554,152.789
C06903=1088.286,-30.598,445.395,174.689,17.555,152.789
C06904=1088.293,-30.349,445.381,174.691,17.556,152.789
C06905=1088.299,-30.099,445.369,174.692,17.558,152.789
C06906=1088.304,-29.849,445.356,174.694,17.560,152.789
C06907=1088.310,-29.599,445.344,174.696,17.562,152.789
C06908=1088.316,-29.350,445.332,174.698,17.563,152.789
C06909=1088.322,-29.101,445.318,174.699,17.564,152.789
C06910=1088.328,-28.851,445.306,174.700,17.566,152.789
C06911=1088.334,-28.601,445.293,174.702,17.567,152.789
C06912=1088.340,-28.352,445.281,174.703,17.569,152.789
C06913=1088.346,-28.102,445.269,174.705,17.570,152.789
C06914=1088.352,-27.853,445.256,174.707,17.572,152.789
C06915=1088.358,-27.603,445.243,174.709,17.573,152.789
C06916=1088.364,-27.353,445.231,174.710,17.575,152.789
C06917=1088.370,-27.103,445.218,174.711,17.577,152.789
C06918=1088.376,-26.854,445.205,174.713,17.578,152.789
C06919=1088.382,-26.604,445.192,174.714,17.580,152.789
C06920=1088.388,-26.354,445.180,174.717,17.581,152.789
C06921=1088.393,-26.106,445.166,174.718,17.583,152.789
C06922=1088.398,-25.856,445.154,174.719,17.585,152.789
C06923=1088.404,-25.606,445.141,174.721,17.586,152.789
C06924=1088.410,-25.356,445.129,174.722,17.588,152.789
C06925=1088.416,-25.107,445.115,174.724,17.589,152.789
C06926=1088.422,-24.857,445.103,174.726,17.591,152.789
C06927=1088.428,-24.608,445.091,174.727,17.593,152.789
C06928=1088.434,-24.358,445.077,174.729,17.594,152.789
C06929=1088.439,-24.108,445.064,174.730,17.596,152.789
C06930=1088.445,-23.858,445.052,174.732,17.597,152.789
C06931=1088.451,-23.609,445.038,174.734,17.599,152.789
C06932=1088.456,-23.360,445.026,174.735,17.601,152.789
C06933=1088.462,-23.110,445.014,174.737,17.602,152.789
C06934=1088.469,-22.861,445.000,174.738,17.604,152.789
C06935=1088.475,-22.611,444.988,174.740,17.605,152.789
C06936=1088.480,-22.361,444.974,174.741,17.606,152.789
C06937=1088.486,-22.111,444.961,174.743,17.608,152.789
C06938=1088.492,-21.861,444.949,174.745,17.610,152.789
C06939=1088.498,-21.612,444.935,174.746,17.612,152.789
C06940=1088.504,-21.362,444.923,174.747,17.613,152.789
C06941=1088.510,-21.114,444.910,174.749,17.614,152.789
C06942=1088.515,-20.864,444.897,174.751,17.616,152.789
C06943=1088.521,-20.614,444.884,174.753,17.618,152.789
C06944=1088.527,-20.364,444.871,174.754,17.620,152.789
C06945=1088.533,-20.114,444.859,174.755,17.621,152.789
C06946=1088.539,-19.865,444.845,174.757,17.623,152.789
C06947=1088.545,-19.615,444.833,174.759,17.624,152.789
C06948=1088.550,-19.366,444.819,174.761,17.626,152.789
C06949=1088.556,-19.116,444.806,174.762,17.628,152.789
C06950=1088.562,-18.867,444.793,174.763,17.629,152.789
C06951=1088.568,-18.617,444.780,174.765,17.631,152.789
C06952=1088.575,-18.367,444.767,174.767,17.632,152.789
C06953=1088.579,-18.118,444.754,174.769,17.634,152.789
C06954=1088.585,-17.869,444.741,174.770,17.636,152.789
C06955=1088.591,-17.619,444.729,174.771,17.637,152.789
C06956=1088.597,-17.370,444.715,174.773,17.639,152.789
C06957=1088.604,-17.097,444.701,174.775,17.640,152.789
C06958=1088.610,-16.826,444.687,174.777,17.642,152.789
C06959=1088.617,-16.554,444.672,174.779,17.644,152.789
C06960=1088.623,-16.281,444.658,174.780,17.646,152.789
C06961=1088.629,-16.033,444.645,174.782,17.647,152.789
C06962=1088.634,-15.783,444.632,174.783,17.649,152.789
C06963=1088.641,-15.533,444.619,174.786,17.650,152.789
C06964=1088.647,-15.284,444.606,174.787,17.652,152.789
C06965=1088.652,-15.034,444.593,174.788,17.654,152.789
C06966=1088.658,-14.785,444.579,174.790,17.655,152.789
C06967=1088.663,-14.535,444.566,174.791,17.657,152.789
C06968=1088.670,-14.285,444.553,174.793,17.659,152.789
C06969=1088.676,-14.036,444.540,174.795,17.660,152.789
C06970=1088.681,-13.786,444.527,174.796,17.662,152.789
C06971=1088.687,-13.537,444.513,174.798,17.663,152.789
C06972=1088.693,-13.287,444.499,174.800,17.665,152.789
C06973=1088.699,-13.037,444.487,174.801,17.667,152.789
C06974=1088.705,-12.788,444.474,174.803,17.668,152.789
C06975=1088.710,-12.538,444.460,174.804,17.670,152.789
C06976=1088.716,-12.288,444.447,174.805,17.672,152.789
C06977=1088.722,-12.039,444.433,174.808,17.673,152.789
C06978=1088.728,-11.790,444.420,174.809,17.675,152.789
C06979=1088.733,-11.539,444.407,174.811,17.676,152.789
C06980=1088.739,-11.290,444.394,174.812,17.678,152.789
C06981=1088.746,-11.041,444.380,174.814,17.680,152.789
C06982=1088.751,-10.791,444.367,174.816,17.682,152.789
C06983=1088.757,-10.541,444.354,174.817,17.683,152.789
C06984=1088.762,-10.292,444.340,174.819,17.684,152.789
C06985=1088.769,-10.043,444.327,174.820,17.686,152.789
C06986=1088.774,-9.792,444.314,174.822,17.688,152.789
C06987=1088.780,-9.543,444.300,174.824,17.690,152.789
C06988=1088.785,-9.293,444.287,174.825,17.691,152.789
C06989=1088.792,-9.044,444.273,174.826,17.693,152.790
C06990=1088.798,-8.795,444.260,174.829,17.694,152.789
C06991=1088.803,-8.545,444.247,174.830,17.696,152.789
C06992=1088.809,-8.296,444.234,174.832,17.698,152.789
C06993=1088.815,-8.046,444.220,174.833,17.699,152.790
C06994=1088.822,-7.796,444.206,174.835,17.701,152.790
C06995=1088.827,-7.546,444.192,174.837,17.703,152.790
C06996=1088.833,-7.297,444.180,174.838,17.704,152.789
C06997=1088.838,-7.047,444.166,174.840,17.706,152.790
C06998=1088.845,-6.798,444.153,174.842,17.708,152.790
C06999=1088.850,-6.548,444.139,174.843,17.709,152.790
C07000=1088.856,-6.299,444.125,174.845,17.711,152.790
C07001=1088.862,-6.049,444.112,174.846,17.712,152.790
C07002=1088.868,-5.800,444.098,174.848,17.714,152.790
C07003=1088.873,-5.550,444.085,174.850,17.716,152.790
C07004=1088.879,-5.301,444.072,174.851,17.717,152.790
C07005=1088.886,-5.050,444.058,174.853,17.719,152.790
C07006=1088.892,-4.801,444.044,174.855,17.721,152.790
C07007=1088.897,-4.551,444.030,174.856,17.722,152.790
C07008=1088.903,-4.302,444.017,174.858,17.724,152.790
C07009=1088.909,-4.053,444.003,174.859,17.725,152.790
C07010=1088.914,-3.803,443.989,174.861,17.727,152.790
C07011=1088.921,-3.554,443.976,174.863,17.729,152.790
C07012=1088.926,-3.304,443.962,174.864,17.730,152.790
C07013=1088.932,-3.055,443.949,174.866,17.732,152.790
C07014=1088.938,-2.805,443.935,174.868,17.734,152.790
C07015=1088.944,-2.555,443.921,174.869,17.735,152.790
C07016=1088.949,-2.305,443.907,174.871,17.737,152.790
C07017=1088.956,-2.056,443.894,174.872,17.738,152.790
C07018=1088.961,-1.806,443.881,174.874,17.741,152.790
C07019=1088.966,-1.556,443.867,174.876,17.742,152.790
C07020=1088.972,-1.307,443.854,174.877,17.744,152.790
C07021=1088.979,-1.034,443.838,174.879,17.746,152.790
C07022=1088.985,-0.760,443.822,174.881,17.747,152.790
C07023=1088.991,-0.487,443.807,174.883,17.750,152.790
C07024=1088.998,-0.213,443.793,174.884,17.751,152.790
C07025=1089.003,0.036,443.779,174.886,17.753,152.790
C07026=1089.009,0.286,443.765,174.888,17.754,152.790
C07027=1089.014,0.535,443.751,174.890,17.756,152.790
C07028=1089.020,0.785,443.738,174.891,17.757,152.790
C07029=1089.026,1.034,443.724,174.892,17.759,152.790
C07030=1089.032,1.285,443.710,174.895,17.761,152.790
C07031=1089.037,1.534,443.696,174.896,17.763,152.790
C07032=1089.044,1.783,443.682,174.897,17.764,152.790
C07033=1089.049,2.032,443.668,174.899,17.766,152.790
C07034=1089.055,2.282,443.654,174.901,17.768,152.790
C07035=1089.060,2.531,443.640,174.903,17.769,152.790
C07036=1089.066,2.781,443.626,174.904,17.771,152.790
C07037=1089.072,3.031,443.613,174.906,17.773,152.790
C07038=1089.078,3.281,443.599,174.907,17.774,152.790
C07039=1089.083,3.530,443.585,174.909,17.776,152.790
C07040=1089.089,3.779,443.570,174.910,17.778,152.790
C07041=1089.095,4.029,443.557,174.913,17.779,152.790
C07042=1089.101,4.279,443.542,174.914,17.781,152.790
C07043=1089.107,4.528,443.529,174.916,17.782,152.790
C07044=1089.112,4.778,443.515,174.918,17.784,152.790
C07045=1089.118,5.027,443.501,174.919,17.786,152.790
C07046=1089.124,5.276,443.487,174.920,17.788,152.790
C07047=1089.130,5.527,443.473,174.922,17.789,152.790
C07048=1089.135,5.776,443.459,174.924,17.791,152.790
C07049=1089.141,6.025,443.445,174.926,17.792,152.790
C07050=1089.147,6.274,443.431,174.927,17.794,152.790
C07051=1089.153,6.524,443.417,174.929,17.796,152.790
C07052=1089.159,6.774,443.403,174.931,17.798,152.790
C07053=1089.164,7.024,443.389,174.932,17.799,152.790
C07054=1089.170,7.273,443.374,174.934,17.800,152.790
C07055=1089.176,7.522,443.361,174.936,17.802,152.790
C07056=1089.182,7.772,443.347,174.937,17.804,152.790
C07057=1089.188,8.022,443.333,174.939,17.806,152.790
C07058=1089.194,8.271,443.318,174.941,17.808,152.790
C07059=1089.199,8.520,443.304,174.943,17.809,152.790
C07060=1089.205,8.771,443.290,174.944,17.810,152.790
C07061=1089.211,9.020,443.276,174.945,17.812,152.790
C07062=1089.216,9.269,443.262,174.948,17.814,152.790
C07063=1089.223,9.520,443.248,174.949,17.816,152.791
C07064=1089.229,9.768,443.234,174.951,17.817,152.790
C07065=1089.235,10.018,443.220,174.953,17.819,152.790
C07066=1089.240,10.267,443.206,174.954,17.820,152.790
C07067=1089.246,10.517,443.191,174.956,17.822,152.791
C07068=1089.252,10.767,443.177,174.958,17.824,152.791
C07069=1089.257,11.016,443.163,174.959,17.825,152.790
C07070=1089.264,11.266,443.148,174.961,17.827,152.790
C07071=1089.269,11.515,443.134,174.962,17.828,152.791
C07072=1089.275,11.764,443.120,174.964,17.831,152.791
C07073=1089.281,12.015,443.106,174.966,17.832,152.791
C07074=1089.287,12.264,443.091,174.967,17.833,152.790
C07075=1089.293,12.513,443.078,174.970,17.835,152.790
C07076=1089.299,12.763,443.063,174.971,17.837,152.791
C07077=1089.305,13.012,443.049,174.972,17.838,152.791
C07078=1089.310,13.262,443.035,174.975,17.840,152.790
C07079=1089.317,13.511,443.020,174.976,17.842,152.790
C07080=1089.322,13.761,443.006,174.978,17.843,152.791
C07081=1089.329,14.010,442.991,174.979,17.845,152.791
C07082=1089.334,14.260,442.977,174.982,17.846,152.790
C07083=1089.340,14.509,442.963,174.983,17.848,152.790
C07084=1089.346,14.759,442.949,174.984,17.850,152.791
C07085=1089.352,15.034,442.932,174.987,17.852,152.791
C07086=1089.358,15.310,442.917,174.989,17.854,152.791
C07087=1089.365,15.585,442.901,174.990,17.855,152.791
C07088=1089.371,15.861,442.885,174.992,17.858,152.791
C07089=1089.377,16.110,442.870,174.994,17.859,152.790
C07090=1089.383,16.360,442.856,174.995,17.860,152.791
C07091=1089.388,16.609,442.841,174.998,17.862,152.791
C07092=1089.394,16.859,442.827,174.999,17.864,152.791
C07093=1089.400,17.108,442.812,175.000,17.865,152.791
C07094=1089.405,17.358,442.799,175.003,17.868,152.791
C07095=1089.412,17.608,442.784,175.004,17.869,152.791
C07096=1089.417,17.856,442.769,175.006,17.870,152.791
C07097=1089.423,18.107,442.755,175.008,17.872,152.791
C07098=1089.428,18.356,442.740,175.009,17.874,152.791
C07099=1089.434,18.606,442.726,175.011,17.875,152.791
C07100=1089.440,18.855,442.711,175.013,17.877,152.791
C07101=1089.446,19.104,442.696,175.014,17.879,152.791
C07102=1089.452,19.354,442.682,175.016,17.880,152.791
C07103=1089.458,19.603,442.667,175.018,17.882,152.791
C07104=1089.463,19.853,442.652,175.020,17.883,152.791
C07105=1089.469,20.103,442.638,175.021,17.885,152.791
C07106=1089.475,20.352,442.623,175.023,17.887,152.791
C07107=1089.481,20.602,442.608,175.025,17.889,152.791
C07108=1089.487,20.851,442.595,175.026,17.890,152.791
C07109=1089.492,21.100,442.579,175.029,17.892,152.791
C07110=1089.498,21.350,442.564,175.030,17.893,152.791
C07111=1089.504,21.600,442.551,175.031,17.895,152.791
C07112=1089.509,21.850,442.535,175.034,17.897,152.791
C07113=1089.515,22.099,442.520,175.035,17.898,152.791
C07114=1089.521,22.348,442.506,175.037,17.900,152.791
C07115=1089.527,22.598,442.492,175.039,17.902,152.791
C07116=1089.532,22.847,442.477,175.040,17.904,152.791
C07117=1089.538,23.097,442.462,175.042,17.905,152.791
C07118=1089.544,23.346,442.447,175.044,17.907,152.791
C07119=1089.549,23.596,442.433,175.045,17.908,152.791
C07120=1089.555,23.845,442.418,175.047,17.910,152.791
C07121=1089.561,24.094,442.403,175.049,17.912,152.791
C07122=1089.567,24.344,442.388,175.051,17.913,152.791
C07123=1089.572,24.594,442.374,175.052,17.915,152.791
C07124=1089.578,24.843,442.359,175.054,17.917,152.791
C07125=1089.584,25.092,442.344,175.056,17.918,152.791
C07126=1089.590,25.342,442.329,175.057,17.919,152.791
C07127=1089.596,25.591,442.314,175.060,17.922,152.791
C07128=1089.602,25.841,442.299,175.061,17.923,152.791
C07129=1089.607,26.091,442.285,175.062,17.925,152.791
C07130=1089.613,26.340,442.270,175.065,17.926,152.791
C07131=1089.619,26.589,442.255,175.066,17.928,152.791
C07132=1089.625,26.839,442.239,175.068,17.929,152.791
C07133=1089.630,27.088,442.225,175.070,17.931,152.791
C07134=1089.637,27.338,442.210,175.071,17.933,152.791
C07135=1089.642,27.587,442.195,175.074,17.935,152.791
C07136=1089.648,27.837,442.180,175.075,17.936,152.791
C07137=1089.653,28.086,442.165,175.077,17.937,152.791
C07138=1089.659,28.336,442.150,175.079,17.940,152.791
C07139=1089.665,28.585,442.136,175.080,17.941,152.791
C07140=1089.671,28.835,442.120,175.082,17.942,152.791
C07141=1089.677,29.084,442.106,175.084,17.944,152.791
C07142=1089.682,29.334,442.090,175.086,17.946,152.791
C07143=1089.688,29.583,442.076,175.087,17.947,152.791
C07144=1089.694,29.833,442.060,175.089,17.949,152.791
C07145=1089.699,30.082,442.045,175.091,17.951,152.791
C07146=1089.705,30.332,442.030,175.093,17.953,152.791
C07147=1089.711,30.581,442.015,175.094,17.954,152.791
C07148=1089.716,30.831,442.000,175.096,17.955,152.791
C07149=1089.723,31.108,441.984,175.098,17.958,152.791
C07150=1089.729,31.385,441.967,175.101,17.960,152.791
C07151=1089.736,31.661,441.949,175.102,17.961,152.791
C07152=1089.742,31.939,441.933,175.104,17.963,152.791
C07153=1089.747,32.187,441.918,175.106,17.964,152.790
C07154=1089.753,32.437,441.902,175.108,17.966,152.790
C07155=1089.759,32.686,441.888,175.109,17.968,152.791
C07156=1089.765,32.936,441.872,175.111,17.969,152.790
C07157=1089.770,33.185,441.858,175.113,17.971,152.790
C07158=1089.776,33.435,441.842,175.115,17.973,152.791
C07159=1089.782,33.685,441.827,175.116,17.974,152.790
C07160=1089.787,33.934,441.812,175.119,17.976,152.790
C07161=1089.794,34.183,441.796,175.120,17.978,152.790
C07162=1089.799,34.433,441.781,175.122,17.980,152.790
C07163=1089.805,34.682,441.766,175.124,17.981,152.790
C07164=1089.811,34.932,441.751,175.125,17.982,152.790
C07165=1089.816,35.181,441.736,175.127,17.984,152.790
C07166=1089.823,35.431,441.721,175.129,17.986,152.790
C07167=1089.828,35.680,441.705,175.131,17.988,152.790
C07168=1089.834,35.930,441.691,175.133,17.989,152.790
C07169=1089.840,36.179,441.674,175.134,17.990,152.790
C07170=1089.845,36.429,441.659,175.137,17.992,152.790
C07171=1089.851,36.678,441.644,175.138,17.993,152.790
C07172=1089.856,36.928,441.629,175.140,17.995,152.790
C07173=1089.863,37.177,441.614,175.142,17.997,152.790
C07174=1089.869,37.427,441.598,175.143,17.998,152.790
C07175=1089.874,37.676,441.583,175.146,18.000,152.790
C07176=1089.880,37.925,441.568,175.147,18.002,152.790
C07177=1089.886,38.175,441.552,175.149,18.003,152.790
C07178=1089.891,38.424,441.536,175.151,18.005,152.790
C07179=1089.898,38.674,441.521,175.152,18.007,152.790
C07180=1089.903,38.923,441.506,175.155,18.008,152.790
C07181=1089.908,39.173,441.491,175.156,18.010,152.790
C07182=1089.914,39.422,441.474,175.158,18.011,152.790
C07183=1089.920,39.671,441.460,175.160,18.013,152.790
C07184=1089.926,39.921,441.444,175.161,18.015,152.790
C07185=1089.931,40.171,441.429,175.164,18.017,152.790
C07186=1089.937,40.420,441.413,175.165,18.018,152.790
C07187=1089.943,40.670,441.398,175.167,18.019,152.790
C07188=1089.948,40.919,441.383,175.169,18.021,152.790
C07189=1089.954,41.168,441.366,175.171,18.023,152.790
C07190=1089.960,41.418,441.351,175.173,18.025,152.790
C07191=1089.965,41.667,441.336,175.174,18.026,152.790
C07192=1089.971,41.916,441.320,175.176,18.027,152.790
C07193=1089.977,42.166,441.304,175.178,18.029,152.790
C07194=1089.982,42.416,441.289,175.180,18.031,152.790
C07195=1089.988,42.665,441.273,175.182,18.033,152.790
C07196=1089.994,42.915,441.257,175.184,18.034,152.790
C07197=1090.000,43.164,441.242,175.186,18.036,152.790
C07198=1090.005,43.413,441.227,175.187,18.037,152.790
C07199=1090.011,43.663,441.211,175.189,18.038,152.790
C07200=1090.017,43.913,441.195,175.191,18.041,152.790
C07201=1090.022,44.162,441.180,175.193,18.042,152.790
C07202=1090.028,44.411,441.163,175.195,18.044,152.790
C07203=1090.034,44.661,441.148,175.196,18.045,152.790
C07204=1090.039,44.910,441.132,175.198,18.046,152.790
C07205=1090.045,45.160,441.116,175.200,18.049,152.790
C07206=1090.050,45.410,441.101,175.202,18.050,152.790
C07207=1090.056,45.658,441.085,175.204,18.052,152.790
C07208=1090.061,45.908,441.069,175.206,18.053,152.790
C07209=1090.067,46.158,441.053,175.208,18.055,152.790
C07210=1090.072,46.407,441.038,175.209,18.056,152.790
C07211=1090.078,46.656,441.022,175.211,18.058,152.790
C07212=1090.084,46.906,441.006,175.213,18.060,152.789
C07213=1090.090,47.183,440.989,175.215,18.062,152.789
C07214=1090.097,47.459,440.971,175.217,18.063,152.789
C07215=1090.103,47.736,440.954,175.219,18.065,152.789
C07216=1090.109,48.014,440.936,175.222,18.067,152.789
C07217=1090.114,48.262,440.920,175.223,18.069,152.789
C07218=1090.120,48.512,440.905,175.225,18.070,152.789
C07219=1090.126,48.762,440.888,175.227,18.072,152.789
C07220=1090.132,49.011,440.872,175.229,18.073,152.789
C07221=1090.137,49.260,440.857,175.231,18.075,152.789
C07222=1090.143,49.510,440.841,175.232,18.077,152.789
C07223=1090.148,49.760,440.825,175.235,18.078,152.789
C07224=1090.154,50.009,440.809,175.236,18.080,152.789
C07225=1090.160,50.258,440.793,175.238,18.081,152.789
C07226=1090.165,50.508,440.777,175.240,18.083,152.789
C07227=1090.171,50.757,440.761,175.242,18.085,152.789
C07228=1090.177,51.006,440.745,175.244,18.086,152.789
C07229=1090.182,51.256,440.730,175.245,18.087,152.789
C07230=1090.188,51.505,440.713,175.248,18.089,152.789
C07231=1090.194,51.754,440.697,175.249,18.090,152.789
C07232=1090.200,52.004,440.682,175.252,18.092,152.789
C07233=1090.206,52.254,440.665,175.253,18.094,152.789
C07234=1090.211,52.502,440.650,175.255,18.096,152.789
C07235=1090.217,52.752,440.634,175.257,18.097,152.789
C07236=1090.222,53.002,440.617,175.259,18.099,152.789
C07237=1090.228,53.251,440.601,175.261,18.100,152.789
C07238=1090.234,53.501,440.585,175.262,18.101,152.789
C07239=1090.240,53.751,440.569,175.265,18.103,152.789
C07240=1090.245,53.999,440.553,175.266,18.105,152.789
C07241=1090.251,54.249,440.537,175.269,18.106,152.788
C07242=1090.257,54.499,440.521,175.270,18.108,152.788
C07243=1090.262,54.748,440.505,175.273,18.109,152.788
C07244=1090.268,54.997,440.489,175.274,18.111,152.788
C07245=1090.274,55.247,440.473,175.276,18.113,152.788
C07246=1090.279,55.496,440.456,175.278,18.114,152.788
C07247=1090.285,55.746,440.441,175.279,18.115,152.788
C07248=1090.291,55.995,440.424,175.282,18.117,152.788
C07249=1090.297,56.244,440.408,175.283,18.118,152.788
C07250=1090.302,56.494,440.392,175.286,18.120,152.788
C07251=1090.308,56.743,440.376,175.287,18.122,152.788
C07252=1090.314,56.992,440.359,175.290,18.123,152.788
C07253=1090.320,57.242,440.344,175.291,18.125,152.788
C07254=1090.325,57.492,440.327,175.294,18.126,152.788
C07255=1090.331,57.741,440.311,175.295,18.127,152.788
C07256=1090.337,57.990,440.295,175.297,18.130,152.788
C07257=1090.342,58.239,440.278,175.299,18.131,152.788
C07258=1090.348,58.489,440.262,175.301,18.133,152.788
C07259=1090.354,58.738,440.246,175.303,18.134,152.788
C07260=1090.360,58.988,440.229,175.305,18.135,152.787
C07261=1090.366,59.237,440.213,175.307,18.137,152.788
C07262=1090.371,59.486,440.197,175.309,18.138,152.787
C07263=1090.377,59.736,440.180,175.311,18.140,152.787
C07264=1090.383,59.985,440.164,175.312,18.141,152.787
C07265=1090.389,60.235,440.149,175.315,18.143,152.787
C07266=1090.394,60.485,440.132,175.317,18.144,152.787
C07267=1090.400,60.734,440.115,175.319,18.146,152.787
C07268=1090.406,60.983,440.099,175.320,18.147,152.787
C07269=1090.412,61.233,440.083,175.323,18.149,152.787
C07270=1090.418,61.482,440.067,175.324,18.150,152.787
C07271=1090.423,61.732,440.050,175.327,18.152,152.787
C07272=1090.429,61.981,440.034,175.328,18.153,152.787
C07273=1090.435,62.230,440.017,175.331,18.155,152.787
C07274=1090.441,62.479,440.000,175.332,18.156,152.787
C07275=1090.447,62.729,439.984,175.334,18.157,152.787
C07276=1090.453,62.978,439.967,175.337,18.159,152.786
C07277=1090.459,63.255,439.950,175.339,18.161,152.786
C07278=1090.465,63.531,439.931,175.340,18.162,152.786
C07279=1090.472,63.808,439.913,175.343,18.164,152.786
C07280=1090.478,64.085,439.895,175.345,18.166,152.786
C07281=1090.484,64.334,439.878,175.347,18.167,152.786
C07282=1090.490,64.583,439.861,175.349,18.168,152.786
C07283=1090.495,64.833,439.845,175.351,18.170,152.786
C07284=1090.501,65.082,439.828,175.353,18.172,152.786
C07285=1090.507,65.332,439.812,175.355,18.173,152.786
C07286=1090.513,65.581,439.795,175.357,18.174,152.786
